C01786=1016.272,-4.523,-107.561,165.907,56.425,160.161
C01787=1016.266,-4.773,-107.549,165.903,56.433,160.162
C01788=1016.261,-5.023,-107.536,165.902,56.442,160.163
C01789=1016.255,-5.301,-107.522,165.899,56.451,160.164
C01790=1016.250,-5.580,-107.508,165.896,56.459,160.165
C01791=1016.243,-5.858,-107.494,165.893,56.468,160.166
C01792=1016.237,-6.136,-107.480,165.889,56.476,160.166
C01793=1016.232,-6.386,-107.466,165.887,56.484,160.167
C01794=1016.226,-6.636,-107.454,165.885,56.492,160.168
C01795=1016.221,-6.886,-107.441,165.882,56.500,160.169
C01796=1016.216,-7.135,-107.429,165.880,56.507,160.170
C01797=1016.210,-7.385,-107.416,165.877,56.515,160.171
C01798=1016.205,-7.634,-107.404,165.874,56.523,160.171
C01799=1016.200,-7.884,-107.391,165.871,56.531,160.172
C01800=1016.194,-8.133,-107.379,165.869,56.538,160.173
C01801=1016.190,-8.384,-107.367,165.866,56.546,160.174
C01802=1016.184,-8.633,-107.354,165.864,56.553,160.175
C01803=1016.179,-8.883,-107.341,165.860,56.561,160.175
C01804=1016.173,-9.133,-107.329,165.858,56.569,160.176
C01805=1016.168,-9.382,-107.317,165.855,56.577,160.177
C01806=1016.164,-9.631,-107.304,165.853,56.584,160.178
C01807=1016.158,-9.881,-107.291,165.850,56.592,160.179
C01808=1016.152,-10.131,-107.279,165.848,56.600,160.180
C01809=1016.147,-10.381,-107.266,165.845,56.607,160.181
C01810=1016.142,-10.630,-107.254,165.842,56.615,160.181
C01811=1016.137,-10.879,-107.242,165.839,56.623,160.182
C01812=1016.131,-11.129,-107.229,165.837,56.630,160.183
C01813=1016.126,-11.379,-107.217,165.834,56.638,160.184
C01814=1016.121,-11.629,-107.204,165.832,56.646,160.185
C01815=1016.116,-11.878,-107.192,165.830,56.653,160.185
C01816=1016.111,-12.128,-107.180,165.827,56.661,160.186
C01817=1016.105,-12.378,-107.166,165.824,56.669,160.187
C01818=1016.100,-12.627,-107.154,165.821,56.677,160.188
C01819=1016.095,-12.876,-107.142,165.819,56.684,160.189
C01820=1016.090,-13.127,-107.130,165.816,56.691,160.189
C01821=1016.085,-13.376,-107.117,165.813,56.699,160.190
C01822=1016.079,-13.625,-107.105,165.811,56.706,160.191
C01823=1016.074,-13.876,-107.092,165.808,56.714,160.192
C01824=1016.069,-14.125,-107.080,165.806,56.722,160.192
C01825=1016.064,-14.374,-107.067,165.803,56.729,160.193
C01826=1016.059,-14.625,-107.055,165.801,56.737,160.194
C01827=1016.053,-14.874,-107.043,165.797,56.744,160.195
C01828=1016.049,-15.123,-107.030,165.795,56.752,160.195
C01829=1016.043,-15.373,-107.018,165.792,56.760,160.196
C01830=1016.038,-15.623,-107.006,165.790,56.767,160.197
C01831=1016.033,-15.873,-106.993,165.787,56.775,160.198
C01832=1016.027,-16.122,-106.981,165.784,56.782,160.198
C01833=1016.022,-16.372,-106.969,165.782,56.790,160.199
C01834=1016.017,-16.621,-106.957,165.779,56.797,160.200
C01835=1016.011,-16.871,-106.945,165.776,56.805,160.201
C01836=1016.006,-17.121,-106.933,165.773,56.813,160.202
C01837=1016.002,-17.371,-106.920,165.771,56.821,160.202
C01838=1015.996,-17.621,-106.909,165.769,56.828,160.203
C01839=1015.991,-17.870,-106.896,165.766,56.836,160.204
C01840=1015.985,-18.120,-106.884,165.764,56.844,160.205
C01841=1015.980,-18.369,-106.873,165.760,56.852,160.206
C01842=1015.975,-18.619,-106.860,165.758,56.859,160.207
C01843=1015.970,-18.869,-106.849,165.755,56.867,160.207
C01844=1015.964,-19.118,-106.837,165.753,56.875,160.208
C01845=1015.959,-19.368,-106.825,165.751,56.882,160.209
C01846=1015.953,-19.618,-106.812,165.747,56.890,160.210
C01847=1015.948,-19.868,-106.801,165.744,56.897,160.210
C01848=1015.943,-20.117,-106.789,165.742,56.905,160.211
C01849=1015.939,-20.367,-106.777,165.739,56.913,160.212
C01850=1015.933,-20.616,-106.765,165.737,56.920,160.213
C01851=1015.928,-20.867,-106.753,165.734,56.928,160.214
C01852=1015.923,-21.116,-106.741,165.732,56.936,160.215
C01853=1015.917,-21.392,-106.727,165.729,56.944,160.215
C01854=1015.911,-21.670,-106.714,165.726,56.952,160.216
C01855=1015.905,-21.946,-106.701,165.722,56.961,160.217
C01856=1015.900,-22.223,-106.688,165.719,56.969,160.218
C01857=1015.894,-22.472,-106.676,165.717,56.977,160.219
C01858=1015.889,-22.722,-106.664,165.714,56.984,160.219
C01859=1015.884,-22.972,-106.652,165.712,56.992,160.220
C01860=1015.879,-23.222,-106.640,165.709,56.999,160.221
C01861=1015.874,-23.471,-106.629,165.707,57.007,160.222
C01862=1015.868,-23.721,-106.617,165.704,57.014,160.222
C01863=1015.863,-23.970,-106.605,165.701,57.022,160.223
C01864=1015.858,-24.220,-106.593,165.699,57.029,160.224
C01865=1015.852,-24.470,-106.581,165.696,57.037,160.225
C01866=1015.847,-24.719,-106.569,165.693,57.044,160.225
C01867=1015.842,-24.969,-106.557,165.690,57.052,160.226
C01868=1015.838,-25.219,-106.545,165.688,57.060,160.227
C01869=1015.832,-25.468,-106.533,165.685,57.067,160.227
C01870=1015.827,-25.718,-106.522,165.682,57.074,160.228
C01871=1015.822,-25.968,-106.510,165.680,57.082,160.229
C01872=1015.817,-26.217,-106.498,165.677,57.089,160.230
C01873=1015.811,-26.468,-106.486,165.675,57.097,160.230
C01874=1015.806,-26.717,-106.474,165.672,57.104,160.231
C01875=1015.801,-26.967,-106.463,165.669,57.111,160.232
C01876=1015.796,-27.216,-106.451,165.667,57.119,160.233
C01877=1015.791,-27.466,-106.439,165.664,57.126,160.233
C01878=1015.786,-27.715,-106.427,165.662,57.134,160.234
C01879=1015.781,-27.965,-106.416,165.659,57.141,160.235
C01880=1015.776,-28.215,-106.404,165.655,57.149,160.235
C01881=1015.771,-28.465,-106.393,165.653,57.156,160.236
C01882=1015.765,-28.714,-106.382,165.651,57.164,160.237
C01883=1015.760,-28.963,-106.370,165.648,57.172,160.238
C01884=1015.755,-29.213,-106.358,165.645,57.179,160.238
C01885=1015.749,-29.464,-106.347,165.643,57.187,160.239
C01886=1015.744,-29.714,-106.335,165.639,57.195,160.240
C01887=1015.738,-29.963,-106.324,165.637,57.202,160.241
C01888=1015.733,-30.213,-106.313,165.634,57.209,160.241
C01889=1015.728,-30.463,-106.301,165.632,57.217,160.242
C01890=1015.723,-30.712,-106.289,165.629,57.225,160.243
C01891=1015.717,-30.961,-106.278,165.627,57.232,160.244
C01892=1015.712,-31.211,-106.267,165.624,57.239,160.245
C01893=1015.707,-31.461,-106.255,165.621,57.248,160.245
C01894=1015.702,-31.711,-106.244,165.618,57.255,160.246
C01895=1015.697,-31.961,-106.232,165.615,57.262,160.247
C01896=1015.692,-32.210,-106.221,165.613,57.270,160.247
C01897=1015.687,-32.460,-106.210,165.611,57.278,160.248
C01898=1015.682,-32.710,-106.199,165.608,57.285,160.249
C01899=1015.677,-32.959,-106.187,165.605,57.292,160.250
C01900=1015.671,-33.209,-106.176,165.602,57.299,160.250
C01901=1015.666,-33.459,-106.165,165.600,57.307,160.251
C01902=1015.661,-33.709,-106.153,165.597,57.315,160.252
C01903=1015.656,-33.958,-106.142,165.594,57.322,160.252
C01904=1015.650,-34.208,-106.131,165.591,57.330,160.253
C01905=1015.645,-34.458,-106.119,165.589,57.337,160.254
C01906=1015.641,-34.707,-106.108,165.586,57.345,160.255
C01907=1015.636,-34.957,-106.097,165.583,57.352,160.255
C01908=1015.631,-35.206,-106.085,165.581,57.359,160.256
C01909=1015.625,-35.456,-106.074,165.578,57.366,160.257
C01910=1015.620,-35.706,-106.063,165.576,57.374,160.257
C01911=1015.615,-35.955,-106.052,165.573,57.381,160.258
C01912=1015.610,-36.205,-106.040,165.570,57.389,160.259
C01913=1015.604,-36.455,-106.029,165.567,57.396,160.259
C01914=1015.599,-36.705,-106.018,165.565,57.403,160.260
C01915=1015.594,-36.954,-106.006,165.562,57.410,160.261
C01916=1015.589,-37.204,-105.995,165.560,57.418,160.262
C01917=1015.584,-37.445,-105.985,165.557,57.425,160.262
C01918=1015.579,-37.685,-105.973,165.554,57.432,160.263
C01919=1015.575,-37.925,-105.963,165.551,57.439,160.263
C01920=1015.570,-38.166,-105.952,165.549,57.447,160.264
C01921=1015.564,-38.406,-105.941,165.547,57.453,160.265
C01922=1015.560,-38.647,-105.930,165.544,57.460,160.266
C01923=1015.555,-38.887,-105.920,165.541,57.467,160.266
C01924=1015.550,-39.128,-105.908,165.538,57.474,160.267
C01925=1015.545,-39.378,-105.898,165.536,57.482,160.267
C01926=1015.540,-39.627,-105.887,165.533,57.489,160.268
C01927=1015.534,-39.877,-105.876,165.531,57.497,160.269
C01928=1015.529,-40.127,-105.864,165.528,57.504,160.269
C01929=1015.524,-40.376,-105.854,165.526,57.512,160.270
C01930=1015.519,-40.626,-105.843,165.523,57.519,160.271
C01931=1015.514,-40.875,-105.832,165.520,57.526,160.272
C01932=1015.509,-41.126,-105.821,165.517,57.535,160.272
C01933=1015.503,-41.375,-105.810,165.514,57.542,160.273
C01934=1015.499,-41.624,-105.799,165.512,57.549,160.274
C01935=1015.493,-41.874,-105.788,165.509,57.556,160.274
C01936=1015.488,-42.124,-105.778,165.507,57.564,160.275
C01937=1015.483,-42.374,-105.767,165.504,57.571,160.276
C01938=1015.478,-42.624,-105.756,165.501,57.579,160.277
C01939=1015.473,-42.873,-105.746,165.498,57.586,160.277
C01940=1015.468,-43.123,-105.734,165.496,57.593,160.278
C01941=1015.462,-43.373,-105.724,165.493,57.601,160.279
C01942=1015.457,-43.623,-105.712,165.490,57.608,160.279
C01943=1015.452,-43.872,-105.702,165.488,57.615,160.280
C01944=1015.448,-44.122,-105.691,165.484,57.623,160.280
C01945=1015.441,-44.416,-105.678,165.481,57.632,160.281
C01946=1015.435,-44.711,-105.665,165.478,57.640,160.282
C01947=1015.430,-45.005,-105.653,165.475,57.649,160.283
C01948=1015.423,-45.299,-105.640,165.472,57.657,160.284
C01949=1015.418,-45.549,-105.630,165.470,57.665,160.284
C01950=1015.413,-45.798,-105.619,165.467,57.672,160.285
C01951=1015.408,-46.048,-105.608,165.464,57.679,160.286
C01952=1015.403,-46.298,-105.597,165.462,57.687,160.286
C01953=1015.397,-46.548,-105.587,165.459,57.694,160.287
C01954=1015.392,-46.797,-105.576,165.456,57.701,160.288
///RCONF 1,0,0,1,0,0,0,0,0,0,0,0,0,0,0,0,0,0,0,0,0,0,0,0
C01955=1015.388,-47.047,-105.565,165.454,57.708,160.288
C01956=1015.382,-47.297,-105.555,165.451,57.715,160.289
C01957=1015.377,-47.546,-105.543,165.448,57.722,160.290
C01958=1015.372,-47.796,-105.533,165.445,57.729,160.290
C01959=1015.367,-48.046,-105.522,165.443,57.737,160.291
C01960=1015.362,-48.295,-105.512,165.440,57.744,160.292
C01961=1015.357,-48.545,-105.501,165.437,57.751,160.292
C01962=1015.352,-48.795,-105.490,165.434,57.758,160.293
C01963=1015.348,-49.045,-105.480,165.432,57.766,160.294
C01964=1015.342,-49.294,-105.469,165.429,57.773,160.294
C01965=1015.337,-49.544,-105.458,165.426,57.780,160.295
C01966=1015.332,-49.793,-105.448,165.423,57.787,160.295
C01967=1015.327,-50.044,-105.437,165.420,57.794,160.296
C01968=1015.322,-50.293,-105.426,165.418,57.802,160.297
C01969=1015.318,-50.543,-105.416,165.415,57.809,160.297
C01970=1015.312,-50.792,-105.405,165.412,57.816,160.298
C01971=1015.307,-51.043,-105.394,165.409,57.823,160.298
C01972=1015.302,-51.292,-105.384,165.407,57.830,160.299
C01973=1015.297,-51.542,-105.374,165.404,57.838,160.300
C01974=1015.291,-51.792,-105.363,165.402,57.845,160.300
C01975=1015.286,-52.041,-105.354,165.399,57.853,160.301
C01976=1015.281,-52.291,-105.343,165.396,57.860,160.302
C01977=1015.275,-52.541,-105.333,165.394,57.868,160.303
C01978=1015.271,-52.791,-105.323,165.391,57.875,160.303
C01979=1015.265,-53.041,-105.313,165.388,57.882,160.304
C01980=1015.260,-53.290,-105.303,165.386,57.889,160.305
C01981=1015.255,-53.566,-105.292,165.383,57.898,160.305
C01982=1015.249,-53.842,-105.280,165.380,57.906,160.306
C01983=1015.243,-54.118,-105.270,165.376,57.914,160.306
C01984=1015.238,-54.394,-105.258,165.374,57.922,160.307
C01985=1015.232,-54.644,-105.248,165.371,57.929,160.308
C01986=1015.227,-54.894,-105.238,165.367,57.936,160.308
C01987=1015.222,-55.144,-105.228,165.365,57.944,160.309
C01988=1015.217,-55.394,-105.218,165.362,57.951,160.310
C01989=1015.212,-55.643,-105.208,165.359,57.958,160.310
C01990=1015.206,-55.894,-105.198,165.357,57.966,160.311
C01991=1015.201,-56.143,-105.188,165.354,57.973,160.312
C01992=1015.196,-56.393,-105.178,165.351,57.980,160.312
C01993=1015.191,-56.642,-105.167,165.349,57.987,160.313
C01994=1015.185,-56.892,-105.157,165.346,57.995,160.314
C01995=1015.181,-57.141,-105.147,165.343,58.002,160.314
C01996=1015.175,-57.391,-105.137,165.341,58.009,160.315
C01997=1015.170,-57.641,-105.127,165.338,58.016,160.315
C01998=1015.165,-57.891,-105.117,165.335,58.023,160.316
C01999=1015.160,-58.140,-105.107,165.333,58.031,160.317
C02000=1015.155,-58.391,-105.096,165.330,58.038,160.317
C02001=1015.151,-58.640,-105.087,165.327,58.045,160.318
C02002=1015.146,-58.890,-105.077,165.324,58.052,160.318
C02003=1015.140,-59.140,-105.067,165.321,58.059,160.319
C02004=1015.135,-59.389,-105.057,165.319,58.067,160.320
C02005=1015.130,-59.639,-105.047,165.316,58.074,160.320
C02006=1015.125,-59.889,-105.037,165.314,58.081,160.321
C02007=1015.120,-60.139,-105.027,165.311,58.088,160.322
C02008=1015.115,-60.388,-105.017,165.308,58.096,160.322
C02009=1015.109,-60.638,-105.007,165.305,58.103,160.323
C02010=1015.105,-60.888,-104.997,165.302,58.110,160.323
C02011=1015.100,-61.137,-104.987,165.299,58.117,160.324
C02012=1015.095,-61.388,-104.978,165.298,58.123,160.325
C02013=1015.090,-61.637,-104.968,165.295,58.130,160.325
C02014=1015.084,-61.887,-104.958,165.292,58.138,160.326
C02015=1015.080,-62.137,-104.948,165.289,58.145,160.326
C02016=1015.075,-62.386,-104.938,165.286,58.152,160.327
C02017=1015.069,-62.636,-104.928,165.284,58.159,160.327
C02018=1015.064,-62.886,-104.918,165.281,58.166,160.328
C02019=1015.059,-63.136,-104.908,165.278,58.173,160.328
C02020=1015.054,-63.385,-104.898,165.275,58.180,160.329
C02021=1015.049,-63.635,-104.889,165.272,58.187,160.330
C02022=1015.044,-63.885,-104.879,165.270,58.194,160.330
C02023=1015.039,-64.135,-104.869,165.268,58.201,160.331
C02024=1015.035,-64.384,-104.860,165.265,58.208,160.331
C02025=1015.029,-64.634,-104.849,165.262,58.215,160.332
C02026=1015.024,-64.884,-104.840,165.259,58.222,160.333
C02027=1015.019,-65.133,-104.830,165.257,58.229,160.333
C02028=1015.015,-65.384,-104.820,165.254,58.236,160.334
C02029=1015.010,-65.633,-104.810,165.251,58.243,160.334
C02030=1015.005,-65.883,-104.800,165.249,58.249,160.335
C02031=1015.000,-66.133,-104.790,165.246,58.256,160.335
C02032=1014.995,-66.382,-104.780,165.243,58.263,160.336
C02033=1014.991,-66.632,-104.771,165.240,58.270,160.336
C02034=1014.986,-66.882,-104.761,165.238,58.278,160.337
C02035=1014.980,-67.132,-104.751,165.235,58.285,160.338
C02036=1014.976,-67.381,-104.741,165.232,58.291,160.338
C02037=1014.971,-67.631,-104.732,165.230,58.298,160.339
C02038=1014.966,-67.882,-104.722,165.227,58.305,160.339
C02039=1014.961,-68.131,-104.712,165.224,58.312,160.340
C02040=1014.956,-68.380,-104.703,165.221,58.319,160.340
C02041=1014.951,-68.630,-104.693,165.219,58.325,160.341
C02042=1014.946,-68.880,-104.683,165.216,58.332,160.341
C02043=1014.941,-69.130,-104.673,165.213,58.339,160.342
C02044=1014.936,-69.379,-104.664,165.210,58.345,160.342
C02045=1014.931,-69.656,-104.653,165.208,58.353,160.343
C02046=1014.926,-69.934,-104.642,165.205,58.360,160.343
C02047=1014.920,-70.210,-104.632,165.201,58.368,160.344
C02048=1014.914,-70.488,-104.621,165.199,58.376,160.345
C02049=1014.909,-70.738,-104.612,165.196,58.382,160.345
C02050=1014.905,-70.987,-104.602,165.193,58.389,160.346
C02051=1014.900,-71.237,-104.592,165.191,58.396,160.346
C02052=1014.895,-71.487,-104.583,165.188,58.402,160.347
C02053=1014.890,-71.737,-104.573,165.185,58.409,160.347
C02054=1014.885,-71.987,-104.564,165.183,58.416,160.348
C02055=1014.881,-72.236,-104.554,165.180,58.422,160.348
C02056=1014.876,-72.486,-104.544,165.177,58.430,160.349
C02057=1014.871,-72.736,-104.535,165.175,58.435,160.349
C02058=1014.866,-72.986,-104.525,165.172,58.443,160.350
C02059=1014.861,-73.235,-104.515,165.169,58.450,160.350
C02060=1014.856,-73.485,-104.506,165.166,58.456,160.350
C02061=1014.852,-73.735,-104.496,165.164,58.463,160.351
C02062=1014.847,-73.985,-104.487,165.161,58.469,160.352
C02063=1014.842,-74.234,-104.477,165.159,58.476,160.352
C02064=1014.837,-74.483,-104.468,165.156,58.482,160.353
C02065=1014.832,-74.734,-104.458,165.153,58.489,160.353
C02066=1014.828,-74.984,-104.449,165.149,58.496,160.353
C02067=1014.823,-75.234,-104.439,165.148,58.502,160.354
C02068=1014.818,-75.484,-104.430,165.145,58.509,160.355
C02069=1014.813,-75.733,-104.421,165.142,58.517,160.355
C02070=1014.808,-75.983,-104.412,165.139,58.523,160.355
C02071=1014.804,-76.233,-104.403,165.137,58.530,160.356
C02072=1014.798,-76.482,-104.394,165.134,58.537,160.357
C02073=1014.794,-76.732,-104.385,165.131,58.543,160.357
C02074=1014.789,-76.982,-104.376,165.128,58.550,160.358
C02075=1014.783,-77.232,-104.366,165.126,58.557,160.358
C02076=1014.778,-77.482,-104.357,165.123,58.563,160.359
C02077=1014.774,-77.732,-104.348,165.120,58.570,160.359
C02078=1014.769,-77.981,-104.338,165.117,58.577,160.359
C02079=1014.764,-78.231,-104.330,165.115,58.583,160.360
C02080=1014.759,-78.481,-104.320,165.113,58.591,160.361
C02081=1014.754,-78.730,-104.311,165.109,58.597,160.361
C02082=1014.749,-78.980,-104.302,165.107,58.604,160.362
C02083=1014.745,-79.230,-104.293,165.104,58.610,160.362
C02084=1014.740,-79.480,-104.284,165.101,58.617,160.363
C02085=1014.735,-79.729,-104.275,165.098,58.624,160.363
C02086=1014.730,-79.979,-104.266,165.096,58.630,160.364
C02087=1014.725,-80.229,-104.257,165.093,58.637,160.364
C02088=1014.721,-80.479,-104.248,165.090,58.644,160.364
C02089=1014.716,-80.729,-104.239,165.089,58.650,160.365
C02090=1014.710,-80.979,-104.231,165.085,58.657,160.365
C02091=1014.706,-81.229,-104.222,165.082,58.664,160.366
C02092=1014.700,-81.478,-104.212,165.080,58.671,160.367
C02093=1014.696,-81.728,-104.203,165.076,58.677,160.367
C02094=1014.691,-81.977,-104.195,165.075,58.684,160.368
C02095=1014.685,-82.227,-104.186,165.072,58.691,160.368
C02096=1014.681,-82.477,-104.177,165.068,58.698,160.368
C02097=1014.675,-82.727,-104.169,165.066,58.705,160.369
C02098=1014.671,-82.977,-104.160,165.063,58.711,160.369
C02099=1014.666,-83.227,-104.151,165.061,58.718,160.370
C02100=1014.661,-83.477,-104.142,165.058,58.725,160.371
C02101=1014.656,-83.726,-104.134,165.056,58.731,160.371
C02102=1014.651,-83.976,-104.125,165.053,58.738,160.372
C02103=1014.646,-84.226,-104.116,165.050,58.745,160.372
C02104=1014.641,-84.476,-104.108,165.047,58.752,160.372
C02105=1014.636,-84.726,-104.098,165.045,58.758,160.373
C02106=1014.632,-84.975,-104.090,165.042,58.765,160.373
C02107=1014.626,-85.225,-104.082,165.038,58.771,160.374
C02108=1014.622,-85.475,-104.073,165.037,58.778,160.374
C02109=1014.616,-85.754,-104.063,165.033,58.786,160.375
C02110=1014.611,-86.033,-104.053,165.030,58.793,160.375
C02111=1014.605,-86.312,-104.044,165.028,58.800,160.376
C02112=1014.600,-86.591,-104.034,165.024,58.807,160.376
C02113=1014.595,-86.841,-104.025,165.022,58.814,160.377
C02114=1014.590,-87.091,-104.017,165.019,58.821,160.377
C02115=1014.585,-87.341,-104.009,165.015,58.827,160.377
C02116=1014.581,-87.590,-104.000,165.014,58.834,160.378
C02117=1014.576,-87.840,-103.992,165.010,58.840,160.378
C02118=1014.571,-88.090,-103.983,165.009,58.847,160.379
C02119=1014.566,-88.340,-103.974,165.005,58.853,160.379
C02120=1014.561,-88.590,-103.966,165.002,58.860,160.380
C02121=1014.556,-88.840,-103.956,165.000,58.866,160.380
C02122=1014.551,-89.089,-103.948,164.997,58.873,160.381
C02123=1014.547,-89.339,-103.939,164.995,58.879,160.381
C02124=1014.542,-89.589,-103.932,164.992,58.886,160.382
C02125=1014.537,-89.839,-103.923,164.990,58.892,160.382
C02126=1014.532,-90.089,-103.914,164.986,58.898,160.382
C02127=1014.527,-90.338,-103.906,164.983,58.905,160.383
C02128=1014.523,-90.588,-103.897,164.981,58.911,160.383
C02129=1014.518,-90.837,-103.888,164.978,58.918,160.384
C02130=1014.513,-91.088,-103.881,164.976,58.924,160.384
C02131=1014.508,-91.338,-103.871,164.973,58.930,160.384
C02132=1014.504,-91.587,-103.863,164.971,58.937,160.385
C02133=1014.499,-91.837,-103.854,164.968,58.943,160.385
C02134=1014.494,-92.087,-103.846,164.965,58.949,160.386
C02135=1014.489,-92.337,-103.838,164.962,58.956,160.386
C02136=1014.485,-92.586,-103.829,164.960,58.962,160.387
C02137=1014.480,-92.836,-103.821,164.957,58.969,160.387
C02138=1014.475,-93.086,-103.812,164.955,58.975,160.388
C02139=1014.470,-93.336,-103.804,164.951,58.981,160.388
C02140=1014.465,-93.585,-103.796,164.949,58.987,160.388
C02141=1014.461,-93.835,-103.787,164.947,58.993,160.389
C02142=1014.456,-94.086,-103.779,164.944,59.000,160.389
C02143=1014.452,-94.335,-103.770,164.941,59.006,160.389
C02144=1014.447,-94.585,-103.762,164.938,59.012,160.390
C02145=1014.442,-94.834,-103.753,164.936,59.018,160.390
C02146=1014.438,-95.084,-103.745,164.933,59.025,160.391
C02147=1014.433,-95.334,-103.737,164.931,59.031,160.391
C02148=1014.427,-95.584,-103.728,164.928,59.037,160.392
C02149=1014.423,-95.834,-103.720,164.925,59.044,160.392
C02150=1014.418,-96.083,-103.712,164.923,59.050,160.392
C02151=1014.414,-96.334,-103.703,164.920,59.056,160.393
C02152=1014.410,-96.583,-103.695,164.917,59.062,160.393
C02153=1014.404,-96.833,-103.687,164.915,59.068,160.393
C02154=1014.400,-97.083,-103.678,164.912,59.074,160.394
C02155=1014.395,-97.333,-103.670,164.909,59.080,160.394
C02156=1014.391,-97.583,-103.661,164.907,59.086,160.395
C02157=1014.386,-97.833,-103.654,164.903,59.092,160.394
C02158=1014.381,-98.082,-103.645,164.901,59.098,160.395
C02159=1014.376,-98.332,-103.638,164.898,59.105,160.396
C02160=1014.372,-98.582,-103.629,164.896,59.111,160.396
C02161=1014.367,-98.832,-103.621,164.893,59.118,160.396
C02162=1014.362,-99.082,-103.613,164.890,59.124,160.397
C02163=1014.357,-99.332,-103.605,164.888,59.130,160.397
C02164=1014.353,-99.581,-103.597,164.885,59.136,160.397
C02165=1014.348,-99.831,-103.589,164.883,59.142,160.398
C02166=1014.343,-100.081,-103.582,164.879,59.149,160.398
C02167=1014.338,-100.331,-103.573,164.877,59.155,160.399
C02168=1014.334,-100.580,-103.566,164.874,59.161,160.399
C02169=1014.328,-100.830,-103.557,164.872,59.167,160.399
C02170=1014.324,-101.081,-103.549,164.869,59.173,160.400
C02171=1014.320,-101.330,-103.541,164.866,59.179,160.400
C02172=1014.315,-101.580,-103.533,164.864,59.185,160.400
C02173=1014.310,-101.861,-103.525,164.861,59.193,160.401
C02174=1014.304,-102.142,-103.516,164.858,59.199,160.401
C02175=1014.299,-102.423,-103.507,164.855,59.206,160.402
C02176=1014.293,-102.704,-103.498,164.852,59.213,160.402
C02177=1014.288,-102.953,-103.490,164.850,59.219,160.402
C02178=1014.284,-103.204,-103.482,164.846,59.225,160.403
C02179=1014.279,-103.453,-103.475,164.844,59.231,160.403
C02180=1014.275,-103.703,-103.466,164.842,59.237,160.404
C02181=1014.270,-103.953,-103.458,164.838,59.244,160.404
C02182=1014.265,-104.203,-103.450,164.836,59.250,160.404
C02183=1014.261,-104.453,-103.443,164.834,59.256,160.405
C02184=1014.256,-104.703,-103.435,164.831,59.262,160.405
C02185=1014.251,-104.952,-103.427,164.828,59.267,160.405
C02186=1014.246,-105.203,-103.419,164.826,59.273,160.405
C02187=1014.242,-105.452,-103.412,164.822,59.280,160.406
C02188=1014.237,-105.702,-103.404,164.820,59.286,160.406
C02189=1014.232,-105.952,-103.396,164.818,59.292,160.407
C02190=1014.228,-106.201,-103.389,164.816,59.298,160.407
C02191=1014.223,-106.452,-103.381,164.812,59.304,160.407
C02192=1014.218,-106.701,-103.373,164.809,59.310,160.407
C02193=1014.213,-106.951,-103.365,164.807,59.316,160.408
C02194=1014.209,-107.201,-103.358,164.805,59.322,160.408
C02195=1014.204,-107.451,-103.350,164.801,59.327,160.408
C02196=1014.200,-107.701,-103.343,164.799,59.333,160.409
C02197=1014.195,-107.950,-103.335,164.797,59.339,160.409
C02198=1014.190,-108.201,-103.327,164.794,59.345,160.410
C02199=1014.186,-108.450,-103.319,164.792,59.351,160.410
C02200=1014.181,-108.700,-103.311,164.788,59.357,160.410
C02201=1014.176,-108.950,-103.304,164.786,59.363,160.410
C02202=1014.172,-109.199,-103.297,164.784,59.369,160.411
C02203=1014.167,-109.450,-103.289,164.781,59.375,160.411
C02204=1014.163,-109.699,-103.281,164.778,59.381,160.411
C02205=1014.158,-109.950,-103.274,164.775,59.387,160.412
C02206=1014.153,-110.199,-103.267,164.773,59.393,160.412
C02207=1014.148,-110.448,-103.259,164.771,59.399,160.413
C02208=1014.143,-110.699,-103.252,164.767,59.405,160.413
C02209=1014.139,-110.948,-103.244,164.765,59.411,160.413
C02210=1014.135,-111.198,-103.237,164.763,59.417,160.413
C02211=1014.130,-111.448,-103.229,164.760,59.422,160.414
C02212=1014.125,-111.698,-103.222,164.757,59.428,160.414
C02213=1014.121,-111.948,-103.214,164.755,59.434,160.415
C02214=1014.115,-112.198,-103.207,164.751,59.440,160.414
C02215=1014.111,-112.447,-103.200,164.749,59.446,160.415
C02216=1014.107,-112.697,-103.192,164.747,59.452,160.415
C02217=1014.102,-112.947,-103.185,164.744,59.457,160.415
C02218=1014.097,-113.197,-103.177,164.742,59.463,160.416
C02219=1014.093,-113.447,-103.170,164.739,59.468,160.416
C02220=1014.089,-113.697,-103.163,164.737,59.474,160.416
C02221=1014.084,-113.947,-103.155,164.734,59.480,160.417
C02222=1014.080,-114.197,-103.148,164.732,59.486,160.417
C02223=1014.075,-114.446,-103.141,164.728,59.492,160.417
C02224=1014.070,-114.696,-103.133,164.726,59.497,160.417
C02225=1014.065,-114.946,-103.126,164.723,59.503,160.418
C02226=1014.061,-115.196,-103.119,164.720,59.509,160.418
C02227=1014.056,-115.445,-103.111,164.718,59.515,160.418
C02228=1014.051,-115.696,-103.105,164.715,59.520,160.419
C02229=1014.047,-115.946,-103.097,164.713,59.526,160.419
C02230=1014.042,-116.195,-103.090,164.710,59.531,160.419
C02231=1014.038,-116.445,-103.082,164.708,59.537,160.420
C02232=1014.032,-116.695,-103.075,164.705,59.543,160.420
C02233=1014.028,-116.945,-103.069,164.703,59.549,160.420
C02234=1014.024,-117.195,-103.061,164.700,59.554,160.420
C02235=1014.020,-117.444,-103.054,164.698,59.560,160.421
C02236=1014.014,-117.694,-103.047,164.695,59.565,160.421
C02237=1014.009,-117.976,-103.039,164.692,59.572,160.421
C02238=1014.004,-118.257,-103.031,164.689,59.578,160.421
C02239=1013.999,-118.538,-103.023,164.686,59.584,160.422
C02240=1013.994,-118.819,-103.015,164.683,59.591,160.422
C02241=1013.989,-119.069,-103.008,164.681,59.597,160.422
C02242=1013.985,-119.320,-103.001,164.678,59.602,160.423
C02243=1013.980,-119.569,-102.994,164.676,59.608,160.423
C02244=1013.975,-119.819,-102.986,164.673,59.613,160.423
C02245=1013.971,-120.069,-102.980,164.670,59.619,160.423
C02246=1013.966,-120.318,-102.973,164.668,59.625,160.424
C02247=1013.962,-120.568,-102.966,164.665,59.630,160.424
C02248=1013.957,-120.819,-102.959,164.663,59.636,160.424
C02249=1013.953,-121.068,-102.951,164.660,59.641,160.424
C02250=1013.948,-121.318,-102.945,164.657,59.647,160.425
C02251=1013.944,-121.568,-102.938,164.655,59.653,160.425
C02252=1013.939,-121.818,-102.930,164.652,59.658,160.425
C02253=1013.935,-122.068,-102.924,164.649,59.663,160.425
C02254=1013.930,-122.317,-102.917,164.648,59.669,160.426
C02255=1013.926,-122.567,-102.910,164.645,59.674,160.426
C02256=1013.921,-122.817,-102.903,164.643,59.679,160.426
C02257=1013.916,-123.067,-102.895,164.640,59.685,160.426
C02258=1013.912,-123.317,-102.889,164.638,59.691,160.427
C02259=1013.907,-123.567,-102.882,164.635,59.696,160.427
C02260=1013.903,-123.817,-102.875,164.632,59.701,160.427
C02261=1013.898,-124.066,-102.868,164.629,59.707,160.427
C02262=1013.894,-124.317,-102.862,164.627,59.711,160.428
C02263=1013.889,-124.566,-102.854,164.625,59.717,160.428
C02264=1013.885,-124.816,-102.848,164.622,59.723,160.428
C02265=1013.880,-125.066,-102.841,164.619,59.728,160.428
C02266=1013.876,-125.316,-102.834,164.617,59.733,160.428
C02267=1013.871,-125.565,-102.827,164.614,59.739,160.429
C02268=1013.867,-125.816,-102.821,164.612,59.745,160.429
C02269=1013.862,-126.066,-102.815,164.609,59.750,160.429
C02270=1013.858,-126.315,-102.807,164.607,59.755,160.429
C02271=1013.853,-126.565,-102.801,164.604,59.760,160.430
C02272=1013.849,-126.815,-102.794,164.602,59.766,160.430
C02273=1013.844,-127.065,-102.788,164.599,59.771,160.430
C02274=1013.840,-127.315,-102.781,164.596,59.777,160.430
C02275=1013.835,-127.564,-102.774,164.595,59.782,160.431
C02276=1013.831,-127.814,-102.767,164.592,59.787,160.431
C02277=1013.826,-128.064,-102.761,164.589,59.792,160.431
C02278=1013.822,-128.314,-102.754,164.586,59.797,160.431
C02279=1013.818,-128.563,-102.747,164.584,59.802,160.431
C02280=1013.813,-128.813,-102.739,164.582,59.806,160.431
C02281=1013.810,-129.062,-102.730,164.580,59.810,160.431
C02282=1013.807,-129.312,-102.721,164.578,59.813,160.431
C02283=1013.804,-129.562,-102.712,164.575,59.817,160.431
C02284=1013.802,-129.812,-102.701,164.572,59.819,160.431
C02285=1013.799,-130.061,-102.690,164.570,59.821,160.430
C02286=1013.798,-130.311,-102.679,164.568,59.821,160.430
C02287=1013.797,-130.560,-102.666,164.566,59.822,160.429
C02288=1013.796,-130.810,-102.653,164.563,59.822,160.429
C02289=1013.795,-131.060,-102.640,164.561,59.822,160.428
C02290=1013.795,-131.310,-102.626,164.560,59.822,160.427
C02291=1013.794,-131.559,-102.612,164.557,59.821,160.426
C02292=1013.795,-131.809,-102.597,164.555,59.819,160.425
C02293=1013.796,-132.059,-102.581,164.552,59.817,160.424
C02294=1013.797,-132.308,-102.565,164.551,59.814,160.423
C02295=1013.798,-132.558,-102.548,164.549,59.811,160.422
C02296=1013.800,-132.807,-102.530,164.547,59.808,160.421
C02297=1013.802,-133.057,-102.512,164.545,59.803,160.419
C02298=1013.804,-133.307,-102.493,164.543,59.799,160.418
C02299=1013.807,-133.556,-102.473,164.541,59.794,160.416
C02300=1013.810,-133.806,-102.453,164.539,59.788,160.415
C02301=1013.579,-133.832,-102.870,164.519,60.110,160.468
C02302=1013.576,-133.583,-102.890,164.521,60.115,160.470
C02303=1013.574,-133.333,-102.909,164.523,60.119,160.471
C02304=1013.571,-133.083,-102.928,164.526,60.124,160.473
C02305=1013.570,-132.833,-102.947,164.527,60.128,160.474
C02306=1013.568,-132.584,-102.965,164.530,60.131,160.475
C02307=1013.566,-132.334,-102.982,164.530,60.134,160.476
C02308=1013.565,-132.084,-102.997,164.533,60.137,160.478
C02309=1013.564,-131.835,-103.014,164.535,60.139,160.478
C02310=1013.564,-131.585,-103.029,164.538,60.140,160.480
C02311=1013.564,-131.336,-103.043,164.539,60.142,160.480
C02312=1013.565,-131.086,-103.057,164.541,60.142,160.481
C02313=1013.565,-130.836,-103.071,164.544,60.142,160.482
C02314=1013.566,-130.587,-103.083,164.545,60.142,160.482
C02315=1013.568,-130.338,-103.096,164.548,60.141,160.483
C02316=1013.569,-130.088,-103.107,164.550,60.140,160.483
C02317=1013.571,-129.838,-103.119,164.552,60.138,160.484
C02318=1013.574,-129.588,-103.129,164.554,60.137,160.484
C02319=1013.576,-129.338,-103.138,164.558,60.134,160.485
C02320=1013.579,-129.088,-103.148,164.560,60.131,160.485
C02321=1013.583,-128.839,-103.156,164.562,60.127,160.485
C02322=1013.586,-128.590,-103.164,164.563,60.123,160.484
C02323=1013.590,-128.340,-103.171,164.567,60.119,160.485
C02324=1013.595,-128.090,-103.178,164.568,60.114,160.484
C02325=1013.600,-127.841,-103.185,164.571,60.109,160.484
C02326=1013.604,-127.591,-103.191,164.574,60.104,160.484
C02327=1013.608,-127.342,-103.198,164.576,60.099,160.484
C02328=1013.613,-127.092,-103.204,164.579,60.094,160.484
C02329=1013.617,-126.842,-103.211,164.581,60.089,160.484
C02330=1013.622,-126.592,-103.218,164.584,60.084,160.483
C02331=1013.626,-126.342,-103.224,164.587,60.078,160.483
C02332=1013.631,-126.092,-103.230,164.588,60.073,160.483
C02333=1013.635,-125.842,-103.238,164.591,60.068,160.483
C02334=1013.640,-125.593,-103.244,164.594,60.063,160.483
C02335=1013.644,-125.342,-103.251,164.597,60.058,160.483
C02336=1013.648,-125.093,-103.258,164.598,60.053,160.482
C02337=1013.653,-124.843,-103.264,164.601,60.047,160.482
C02338=1013.658,-124.593,-103.272,164.604,60.042,160.482
C02339=1013.662,-124.343,-103.278,164.606,60.037,160.482
C02340=1013.667,-124.093,-103.285,164.608,60.032,160.481
C02341=1013.671,-123.843,-103.292,164.611,60.027,160.481
C02342=1013.677,-123.593,-103.299,164.613,60.022,160.481
C02343=1013.681,-123.343,-103.306,164.616,60.016,160.481
C02344=1013.685,-123.093,-103.313,164.619,60.011,160.481
C02345=1013.690,-122.843,-103.319,164.621,60.006,160.481
C02346=1013.694,-122.594,-103.327,164.623,60.001,160.480
C02347=1013.698,-122.343,-103.333,164.626,59.996,160.480
C02348=1013.703,-122.094,-103.340,164.629,59.990,160.480
C02349=1013.707,-121.844,-103.347,164.632,59.985,160.480
C02350=1013.712,-121.594,-103.354,164.633,59.980,160.479
C02351=1013.716,-121.344,-103.360,164.636,59.975,160.479
C02352=1013.721,-121.095,-103.368,164.638,59.969,160.479
C02353=1013.725,-120.845,-103.375,164.641,59.963,160.479
C02354=1013.731,-120.594,-103.381,164.644,59.958,160.479
C02355=1013.735,-120.345,-103.389,164.646,59.953,160.478
C02356=1013.739,-120.095,-103.396,164.648,59.948,160.478
C02357=1013.744,-119.845,-103.402,164.651,59.943,160.478
C02358=1013.748,-119.596,-103.410,164.654,59.937,160.478
C02359=1013.752,-119.345,-103.416,164.656,59.931,160.477
C02360=1013.757,-119.096,-103.424,164.659,59.926,160.477
C02361=1013.762,-118.846,-103.431,164.662,59.921,160.477
C02362=1013.766,-118.565,-103.438,164.664,59.915,160.477
C02363=1013.772,-118.283,-103.447,164.667,59.908,160.476
C02364=1013.778,-118.002,-103.454,164.670,59.903,160.476
C02365=1013.783,-117.721,-103.463,164.673,59.896,160.476
C02366=1013.787,-117.471,-103.470,164.675,59.891,160.476
C02367=1013.792,-117.222,-103.477,164.677,59.885,160.475
C02368=1013.796,-116.972,-103.483,164.680,59.880,160.475
C02369=1013.800,-116.722,-103.491,164.683,59.875,160.475
C02370=1013.805,-116.472,-103.499,164.685,59.869,160.475
C02371=1013.810,-116.222,-103.506,164.688,59.863,160.474
C02372=1013.815,-115.972,-103.512,164.690,59.858,160.474
C02373=1013.819,-115.723,-103.519,164.693,59.853,160.474
C02374=1013.823,-115.473,-103.527,164.695,59.847,160.474
C02375=1013.828,-115.223,-103.535,164.698,59.841,160.473
C02376=1013.833,-114.973,-103.541,164.700,59.835,160.473
C02377=1013.837,-114.723,-103.548,164.703,59.830,160.473
C02378=1013.842,-114.474,-103.556,164.706,59.825,160.473
C02379=1013.847,-114.223,-103.563,164.708,59.819,160.472
C02380=1013.851,-113.974,-103.571,164.711,59.813,160.472
C02381=1013.855,-113.724,-103.578,164.714,59.808,160.472
C02382=1013.860,-113.475,-103.585,164.716,59.802,160.471
C02383=1013.865,-113.224,-103.592,164.719,59.797,160.471
C02384=1013.869,-112.974,-103.599,164.722,59.791,160.471
C02385=1013.874,-112.724,-103.607,164.724,59.785,160.471
C02386=1013.878,-112.475,-103.614,164.727,59.780,160.471
C02387=1013.883,-112.224,-103.622,164.729,59.774,160.470
C02388=1013.887,-111.975,-103.629,164.732,59.769,160.470
C02389=1013.892,-111.725,-103.637,164.734,59.763,160.469
C02390=1013.896,-111.475,-103.644,164.737,59.757,160.469
C02391=1013.902,-111.225,-103.651,164.739,59.751,160.469
C02392=1013.906,-110.976,-103.659,164.742,59.746,160.469
C02393=1013.911,-110.726,-103.666,164.744,59.740,160.468
C02394=1013.916,-110.476,-103.674,164.747,59.735,160.468
C02395=1013.920,-110.226,-103.681,164.749,59.729,160.468
C02396=1013.924,-109.977,-103.689,164.751,59.723,160.468
C02397=1013.929,-109.726,-103.696,164.754,59.717,160.467
C02398=1013.934,-109.477,-103.704,164.756,59.712,160.467
C02399=1013.939,-109.227,-103.711,164.760,59.705,160.467
C02400=1013.944,-108.977,-103.718,164.763,59.700,160.467
C02401=1013.948,-108.727,-103.726,164.765,59.694,160.466
C02402=1013.952,-108.478,-103.733,164.767,59.688,160.466
C02403=1013.957,-108.227,-103.741,164.770,59.683,160.465
C02404=1013.962,-107.978,-103.748,164.772,59.677,160.465
C02405=1013.967,-107.727,-103.756,164.775,59.671,160.465
C02406=1013.971,-107.478,-103.764,164.777,59.665,160.464
C02407=1013.975,-107.228,-103.771,164.780,59.659,160.464
C02408=1013.980,-106.978,-103.779,164.783,59.654,160.464
C02409=1013.985,-106.728,-103.786,164.785,59.648,160.464
C02410=1013.990,-106.478,-103.795,164.788,59.642,160.463
C02411=1013.994,-106.229,-103.802,164.790,59.636,160.463
C02412=1013.999,-105.979,-103.809,164.792,59.630,160.462
C02413=1014.004,-105.729,-103.817,164.795,59.625,160.462
C02414=1014.008,-105.479,-103.825,164.798,59.619,160.462
C02415=1014.013,-105.229,-103.832,164.801,59.612,160.462
C02416=1014.018,-104.980,-103.841,164.803,59.607,160.461
C02417=1014.022,-104.729,-103.849,164.806,59.601,160.461
C02418=1014.026,-104.480,-103.856,164.808,59.595,160.461
C02419=1014.031,-104.230,-103.864,164.812,59.589,160.461
C02420=1014.036,-103.980,-103.872,164.814,59.583,160.460
C02421=1014.040,-103.731,-103.880,164.816,59.577,160.460
C02422=1014.045,-103.480,-103.887,164.818,59.571,160.459
C02423=1014.049,-103.231,-103.895,164.821,59.566,160.459
C02424=1014.055,-102.981,-103.903,164.824,59.560,160.459
C02425=1014.059,-102.731,-103.911,164.827,59.554,160.458
C02426=1014.065,-102.450,-103.920,164.830,59.547,160.458
C02427=1014.070,-102.169,-103.928,164.832,59.540,160.458
C02428=1014.075,-101.889,-103.937,164.836,59.533,160.457
C02429=1014.081,-101.607,-103.946,164.839,59.527,160.457
C02430=1014.084,-101.357,-103.954,164.841,59.521,160.457
C02431=1014.089,-101.107,-103.962,164.843,59.515,160.456
C02432=1014.094,-100.858,-103.970,164.846,59.509,160.456
C02433=1014.099,-100.608,-103.978,164.849,59.502,160.455
C02434=1014.103,-100.358,-103.985,164.851,59.496,160.455
C02435=1014.109,-100.108,-103.994,164.854,59.491,160.455
C02436=1014.113,-99.859,-104.001,164.857,59.485,160.455
C02437=1014.118,-99.609,-104.010,164.859,59.478,160.454
C02438=1014.123,-99.359,-104.017,164.861,59.472,160.454
C02439=1014.128,-99.109,-104.025,164.865,59.466,160.453
C02440=1014.132,-98.859,-104.034,164.867,59.460,160.453
C02441=1014.136,-98.609,-104.041,164.869,59.454,160.452
C02442=1014.141,-98.359,-104.049,164.872,59.447,160.452
C02443=1014.146,-98.110,-104.057,164.875,59.441,160.452
C02444=1014.151,-97.860,-104.065,164.878,59.435,160.451
C02445=1014.156,-97.610,-104.074,164.880,59.429,160.451
C02446=1014.160,-97.360,-104.082,164.883,59.424,160.451
C02447=1014.165,-97.110,-104.090,164.885,59.418,160.450
C02448=1014.169,-96.861,-104.099,164.888,59.411,160.450
C02449=1014.174,-96.611,-104.107,164.891,59.405,160.450
C02450=1014.179,-96.361,-104.116,164.893,59.399,160.449
C02451=1014.183,-96.111,-104.123,164.896,59.393,160.449
C02452=1014.188,-95.861,-104.132,164.898,59.387,160.448
C02453=1014.193,-95.611,-104.141,164.901,59.381,160.448
C02454=1014.197,-95.362,-104.148,164.903,59.375,160.448
C02455=1014.202,-95.112,-104.156,164.907,59.369,160.448
C02456=1014.207,-94.862,-104.166,164.909,59.363,160.447
C02457=1014.211,-94.612,-104.173,164.911,59.357,160.447
C02458=1014.216,-94.362,-104.182,164.914,59.350,160.446
C02459=1014.221,-94.113,-104.191,164.917,59.344,160.446
C02460=1014.225,-93.863,-104.198,164.920,59.338,160.446
C02461=1014.230,-93.613,-104.207,164.922,59.332,160.445
C02462=1014.235,-93.363,-104.215,164.924,59.326,160.445
C02463=1014.239,-93.113,-104.223,164.928,59.320,160.445
C02464=1014.244,-92.864,-104.232,164.930,59.314,160.444
C02465=1014.249,-92.614,-104.240,164.933,59.307,160.444
C02466=1014.253,-92.365,-104.249,164.935,59.301,160.443
C02467=1014.258,-92.114,-104.257,164.937,59.295,160.443
C02468=1014.263,-91.864,-104.266,164.941,59.289,160.443
C02469=1014.268,-91.614,-104.275,164.943,59.283,160.442
C02470=1014.273,-91.365,-104.283,164.946,59.276,160.442
C02471=1014.277,-91.115,-104.291,164.948,59.269,160.441
C02472=1014.282,-90.865,-104.299,164.951,59.263,160.441
C02473=1014.286,-90.616,-104.308,164.953,59.257,160.440
C02474=1014.291,-90.366,-104.317,164.957,59.251,160.440
C02475=1014.296,-90.116,-104.324,164.959,59.245,160.440
C02476=1014.301,-89.866,-104.334,164.962,59.238,160.439
C02477=1014.306,-89.617,-104.342,164.964,59.232,160.439
C02478=1014.310,-89.367,-104.351,164.967,59.225,160.438
C02479=1014.315,-89.117,-104.359,164.969,59.219,160.438
C02480=1014.320,-88.867,-104.367,164.973,59.212,160.438
C02481=1014.325,-88.617,-104.376,164.975,59.206,160.437
C02482=1014.329,-88.368,-104.384,164.977,59.199,160.437
C02483=1014.334,-88.118,-104.393,164.980,59.193,160.436
C02484=1014.339,-87.868,-104.402,164.983,59.187,160.436
C02485=1014.344,-87.618,-104.410,164.985,59.181,160.435
C02486=1014.349,-87.367,-104.419,164.988,59.174,160.435
C02487=1014.353,-87.118,-104.427,164.990,59.168,160.434
C02488=1014.358,-86.868,-104.436,164.993,59.161,160.434
C02489=1014.363,-86.619,-104.444,164.996,59.154,160.434
C02490=1014.368,-86.340,-104.454,164.999,59.148,160.433
C02491=1014.374,-86.060,-104.464,165.002,59.140,160.433
C02492=1014.380,-85.782,-104.473,165.005,59.133,160.432
C02493=1014.385,-85.503,-104.483,165.008,59.126,160.432
C02494=1014.390,-85.253,-104.491,165.010,59.119,160.431
C02495=1014.395,-85.003,-104.500,165.013,59.112,160.431
C02496=1014.400,-84.754,-104.509,165.016,59.105,160.430
C02497=1014.404,-84.504,-104.518,165.018,59.099,160.430
C02498=1014.409,-84.255,-104.526,165.022,59.093,160.429
C02499=1014.414,-84.005,-104.535,165.023,59.086,160.429
C02500=1014.419,-83.755,-104.543,165.026,59.080,160.428
C02501=1014.424,-83.505,-104.552,165.029,59.072,160.428
C02502=1014.429,-83.255,-104.561,165.031,59.066,160.427
C02503=1014.434,-83.005,-104.569,165.034,59.059,160.427
C02504=1014.438,-82.755,-104.578,165.037,59.053,160.427
C02505=1014.444,-82.506,-104.587,165.040,59.046,160.426
C02506=1014.449,-82.256,-104.595,165.042,59.040,160.425
C02507=1014.453,-82.006,-104.605,165.045,59.033,160.425
C02508=1014.459,-81.756,-104.613,165.048,59.026,160.425
C02509=1014.463,-81.507,-104.622,165.050,59.019,160.424
C02510=1014.468,-81.257,-104.630,165.053,59.012,160.423
C02511=1014.472,-81.007,-104.639,165.056,59.006,160.423
C02512=1014.478,-80.757,-104.648,165.059,58.999,160.422
C02513=1014.483,-80.508,-104.656,165.061,58.993,160.422
C02514=1014.488,-80.258,-104.665,165.063,58.985,160.421
C02515=1014.492,-80.008,-104.674,165.067,58.979,160.421
C02516=1014.497,-79.758,-104.683,165.068,58.972,160.420
C02517=1014.502,-79.508,-104.692,165.072,58.966,160.420
C02518=1014.507,-79.259,-104.702,165.074,58.959,160.420
C02519=1014.511,-79.008,-104.711,165.077,58.953,160.419
C02520=1014.516,-78.759,-104.719,165.080,58.946,160.419
C02521=1014.521,-78.509,-104.728,165.083,58.939,160.418
C02522=1014.526,-78.259,-104.738,165.085,58.933,160.418
C02523=1014.531,-78.010,-104.747,165.088,58.926,160.417
C02524=1014.536,-77.760,-104.756,165.091,58.920,160.417
C02525=1014.540,-77.510,-104.765,165.093,58.913,160.416
C02526=1014.546,-77.260,-104.774,165.095,58.906,160.416
C02527=1014.551,-77.010,-104.783,165.099,58.899,160.415
C02528=1014.555,-76.760,-104.793,165.100,58.893,160.415
C02529=1014.560,-76.510,-104.802,165.104,58.886,160.414
C02530=1014.565,-76.261,-104.811,165.106,58.879,160.414
C02531=1014.570,-76.011,-104.820,165.110,58.873,160.413
C02532=1014.575,-75.761,-104.830,165.111,58.866,160.413
C02533=1014.580,-75.511,-104.838,165.114,58.859,160.412
C02534=1014.585,-75.261,-104.847,165.117,58.852,160.412
C02535=1014.589,-75.012,-104.857,165.120,58.845,160.411
C02536=1014.595,-74.762,-104.866,165.122,58.838,160.410
C02537=1014.599,-74.512,-104.875,165.125,58.832,160.410
C02538=1014.604,-74.263,-104.884,165.128,58.825,160.410
C02539=1014.609,-74.013,-104.894,165.130,58.819,160.409
C02540=1014.614,-73.763,-104.904,165.133,58.812,160.409
C02541=1014.619,-73.513,-104.913,165.136,58.805,160.408
C02542=1014.623,-73.263,-104.923,165.138,58.799,160.408
C02543=1014.628,-73.014,-104.932,165.141,58.792,160.407
C02544=1014.633,-72.764,-104.941,165.143,58.786,160.407
C02545=1014.638,-72.514,-104.951,165.146,58.779,160.406
C02546=1014.642,-72.264,-104.960,165.149,58.772,160.406
C02547=1014.647,-72.015,-104.970,165.152,58.766,160.405
C02548=1014.652,-71.764,-104.980,165.154,58.759,160.405
C02549=1014.657,-71.515,-104.989,165.157,58.753,160.404
C02550=1014.662,-71.265,-104.999,165.160,58.745,160.404
C02551=1014.666,-71.015,-105.008,165.162,58.739,160.403
C02552=1014.671,-70.766,-105.018,165.165,58.732,160.403
C02553=1014.676,-70.517,-105.028,165.167,58.725,160.402
C02554=1014.681,-70.239,-105.039,165.170,58.718,160.402
C02555=1014.687,-69.962,-105.050,165.173,58.711,160.401
C02556=1014.692,-69.685,-105.060,165.177,58.703,160.401
C02557=1014.697,-69.409,-105.071,165.179,58.695,160.400
C02558=1014.701,-69.159,-105.080,165.182,58.689,160.399
C02559=1014.707,-68.908,-105.090,165.185,58.682,160.399
C02560=1014.712,-68.659,-105.100,165.186,58.675,160.398
C02561=1014.716,-68.409,-105.109,165.190,58.669,160.398
C02562=1014.721,-68.160,-105.119,165.193,58.662,160.397
C02563=1014.726,-67.909,-105.129,165.195,58.655,160.397
C02564=1014.731,-67.659,-105.138,165.198,58.649,160.396
C02565=1014.736,-67.410,-105.148,165.200,58.642,160.396
C02566=1014.741,-67.161,-105.158,165.203,58.634,160.395
C02567=1014.745,-66.911,-105.167,165.206,58.627,160.395
C02568=1014.751,-66.661,-105.177,165.209,58.620,160.394
C02569=1014.755,-66.411,-105.187,165.211,58.614,160.393
C02570=1014.760,-66.162,-105.196,165.214,58.607,160.393
C02571=1014.766,-65.912,-105.207,165.216,58.600,160.392
C02572=1014.770,-65.662,-105.216,165.219,58.593,160.392
C02573=1014.775,-65.412,-105.226,165.222,58.586,160.391
C02574=1014.780,-65.163,-105.235,165.225,58.579,160.391
C02575=1014.785,-64.913,-105.245,165.227,58.573,160.390
C02576=1014.790,-64.663,-105.255,165.230,58.566,160.390
C02577=1014.795,-64.413,-105.264,165.232,58.558,160.389
C02578=1014.800,-64.163,-105.275,165.235,58.551,160.388
C02579=1014.805,-63.914,-105.284,165.238,58.544,160.388
C02580=1014.810,-63.664,-105.294,165.240,58.537,160.387
C02581=1014.815,-63.414,-105.304,165.243,58.530,160.387
C02582=1014.820,-63.164,-105.313,165.246,58.523,160.386
C02583=1014.825,-62.915,-105.323,165.248,58.516,160.385
C02584=1014.830,-62.665,-105.333,165.250,58.509,160.385
C02585=1014.835,-62.415,-105.343,165.254,58.503,160.384
C02586=1014.840,-62.166,-105.353,165.257,58.496,160.384
C02587=1014.844,-61.915,-105.363,165.259,58.488,160.383
C02588=1014.849,-61.665,-105.373,165.262,58.481,160.383
C02589=1014.854,-61.416,-105.383,165.265,58.474,160.382
C02590=1014.859,-61.166,-105.393,165.268,58.467,160.382
C02591=1014.864,-60.916,-105.402,165.270,58.459,160.381
C02592=1014.869,-60.667,-105.412,165.272,58.452,160.380
C02593=1014.874,-60.417,-105.422,165.275,58.445,160.380
C02594=1014.879,-60.168,-105.432,165.278,58.438,160.379
C02595=1014.884,-59.917,-105.442,165.281,58.431,160.378
C02596=1014.889,-59.668,-105.452,165.284,58.424,160.378
C02597=1014.894,-59.418,-105.461,165.286,58.417,160.377
C02598=1014.899,-59.168,-105.471,165.289,58.409,160.377
C02599=1014.904,-58.918,-105.481,165.292,58.402,160.376
C02600=1014.910,-58.668,-105.491,165.295,58.395,160.376
C02601=1014.914,-58.419,-105.501,165.297,58.388,160.375
C02602=1014.919,-58.170,-105.511,165.299,58.380,160.374
C02603=1014.925,-57.919,-105.521,165.302,58.373,160.374
C02604=1014.929,-57.670,-105.531,165.305,58.366,160.373
C02605=1014.935,-57.420,-105.541,165.308,58.359,160.372
C02606=1014.940,-57.170,-105.551,165.311,58.352,160.372
C02607=1014.945,-56.920,-105.561,165.313,58.345,160.371
C02608=1014.950,-56.671,-105.571,165.315,58.337,160.370
C02609=1014.955,-56.421,-105.581,165.318,58.330,160.370
C02610=1014.960,-56.171,-105.591,165.321,58.323,160.369
C02611=1014.966,-55.921,-105.601,165.324,58.316,160.369
C02612=1014.970,-55.672,-105.611,165.326,58.308,160.368
C02613=1014.975,-55.422,-105.622,165.329,58.301,160.367
C02614=1014.980,-55.172,-105.631,165.332,58.294,160.367
C02615=1014.986,-54.922,-105.641,165.334,58.287,160.366
C02616=1014.990,-54.673,-105.651,165.336,58.279,160.365
C02617=1014.996,-54.422,-105.661,165.339,58.272,160.365
C02618=1015.001,-54.148,-105.672,165.343,58.263,160.364
C02619=1015.007,-53.872,-105.684,165.346,58.255,160.363
C02620=1015.013,-53.596,-105.694,165.348,58.247,160.362
C02621=1015.019,-53.320,-105.706,165.351,58.239,160.362
C02622=1015.023,-53.070,-105.716,165.354,58.232,160.361
C02623=1015.029,-52.820,-105.726,165.356,58.224,160.360
C02624=1015.034,-52.570,-105.736,165.360,58.217,160.360
C02625=1015.039,-52.321,-105.746,165.362,58.209,160.359
C02626=1015.044,-52.070,-105.756,165.365,58.202,160.358
C02627=1015.049,-51.821,-105.766,165.368,58.195,160.358
C02628=1015.055,-51.572,-105.777,165.370,58.187,160.357
C02629=1015.060,-51.322,-105.787,165.373,58.180,160.356
C02630=1015.065,-51.072,-105.797,165.375,58.172,160.355
C02631=1015.070,-50.822,-105.808,165.378,58.165,160.355
C02632=1015.074,-50.573,-105.819,165.381,58.158,160.354
C02633=1015.080,-50.322,-105.829,165.383,58.151,160.354
C02634=1015.085,-50.072,-105.840,165.386,58.144,160.353
C02635=1015.090,-49.823,-105.850,165.389,58.137,160.353
C02636=1015.094,-49.573,-105.861,165.391,58.129,160.352
C02637=1015.100,-49.324,-105.871,165.394,58.122,160.351
C02638=1015.104,-49.074,-105.882,165.397,58.115,160.351
C02639=1015.110,-48.823,-105.892,165.400,58.108,160.350
C02640=1015.115,-48.575,-105.903,165.402,58.100,160.349
C02641=1015.119,-48.324,-105.914,165.405,58.093,160.349
C02642=1015.125,-48.075,-105.925,165.407,58.086,160.348
C02643=1015.129,-47.825,-105.935,165.410,58.079,160.347
C02644=1015.135,-47.576,-105.946,165.412,58.071,160.347
C02645=1015.140,-47.325,-105.957,165.415,58.064,160.346
C02646=1015.145,-47.076,-105.967,165.418,58.057,160.345
C02647=1015.150,-46.826,-105.978,165.421,58.050,160.345
C02648=1015.155,-46.576,-105.988,165.423,58.042,160.344
///RCONF 1,0,0,0,0,0,0,0,0,0,0,0,0,0,0,0,0,0,0,0,0,0,0,0
C02649=1015.159,-46.327,-105.999,165.426,58.035,160.343
C02650=1015.165,-46.077,-106.009,165.429,58.028,160.343
C02651=1015.170,-45.827,-106.021,165.431,58.020,160.342
C02652=1015.175,-45.578,-106.031,165.434,58.013,160.341
C02653=1015.180,-45.328,-106.042,165.436,58.005,160.340
C02654=1015.185,-45.078,-106.053,165.439,57.998,160.340
C02655=1015.190,-44.828,-106.063,165.443,57.990,160.340
C02656=1015.195,-44.579,-106.074,165.445,57.983,160.339
C02657=1015.201,-44.329,-106.084,165.448,57.976,160.338
C02658=1015.205,-44.080,-106.095,165.450,57.968,160.337
C02659=1015.211,-43.830,-106.106,165.453,57.961,160.337
C02660=1015.216,-43.580,-106.117,165.456,57.954,160.336
C02661=1015.221,-43.330,-106.127,165.458,57.946,160.335
C02662=1015.225,-43.081,-106.138,165.461,57.939,160.335
C02663=1015.231,-42.831,-106.149,165.463,57.931,160.334
C02664=1015.236,-42.581,-106.160,165.466,57.924,160.333
C02665=1015.242,-42.331,-106.171,165.469,57.916,160.332
C02666=1015.246,-42.081,-106.181,165.472,57.909,160.332
C02667=1015.251,-41.832,-106.192,165.474,57.901,160.331
C02668=1015.256,-41.582,-106.204,165.477,57.894,160.330
C02669=1015.262,-41.332,-106.214,165.479,57.886,160.330
C02670=1015.266,-41.083,-106.225,165.482,57.879,160.329
C02671=1015.272,-40.833,-106.236,165.484,57.871,160.328
C02672=1015.277,-40.583,-106.246,165.487,57.864,160.328
C02673=1015.282,-40.334,-106.257,165.490,57.856,160.327
C02674=1015.287,-40.083,-106.268,165.493,57.848,160.326
C02675=1015.292,-39.834,-106.279,165.495,57.841,160.325
C02676=1015.297,-39.585,-106.290,165.498,57.833,160.325
C02677=1015.303,-39.335,-106.301,165.500,57.826,160.324
C02678=1015.308,-39.085,-106.312,165.503,57.819,160.323
C02679=1015.313,-38.835,-106.323,165.506,57.812,160.323
C02680=1015.318,-38.585,-106.335,165.508,57.805,160.322
C02681=1015.323,-38.336,-106.345,165.511,57.797,160.321
C02682=1015.328,-38.061,-106.358,165.514,57.789,160.320
C02683=1015.333,-37.785,-106.370,165.517,57.780,160.320
C02684=1015.339,-37.510,-106.382,165.520,57.773,160.319
C02685=1015.345,-37.234,-106.394,165.523,57.764,160.318
C02686=1015.350,-36.984,-106.406,165.525,57.757,160.317
C02687=1015.355,-36.734,-106.417,165.528,57.750,160.317
C02688=1015.360,-36.484,-106.429,165.530,57.742,160.316
C02689=1015.366,-36.235,-106.439,165.534,57.734,160.315
C02690=1015.371,-35.985,-106.451,165.536,57.727,160.315
C02691=1015.376,-35.735,-106.462,165.539,57.719,160.314
C02692=1015.381,-35.485,-106.474,165.542,57.712,160.313
C02693=1015.386,-35.237,-106.484,165.544,57.704,160.312
C02694=1015.390,-34.986,-106.495,165.547,57.697,160.312
C02695=1015.395,-34.736,-106.507,165.549,57.689,160.311
C02696=1015.400,-34.487,-106.518,165.552,57.682,160.310
C02697=1015.406,-34.237,-106.529,165.554,57.675,160.309
C02698=1015.411,-33.987,-106.540,165.557,57.666,160.309
C02699=1015.416,-33.737,-106.552,165.560,57.659,160.308
C02700=1015.421,-33.488,-106.563,165.563,57.652,160.307
C02701=1015.427,-33.238,-106.574,165.565,57.645,160.307
C02702=1015.435,-32.836,-106.593,165.570,57.632,160.305
C02703=1015.443,-32.432,-106.610,165.574,57.620,160.304
C02704=1015.451,-32.029,-106.629,165.578,57.607,160.303
C02705=1015.459,-31.626,-106.648,165.582,57.595,160.302
C02706=1015.465,-31.376,-106.659,165.585,57.588,160.301
C02707=1015.470,-31.127,-106.670,165.587,57.580,160.300
C02708=1015.475,-30.877,-106.682,165.590,57.572,160.299
C02709=1015.480,-30.627,-106.693,165.593,57.565,160.299
C02710=1015.486,-30.377,-106.704,165.596,57.557,160.298
C02711=1015.491,-30.128,-106.716,165.598,57.549,160.297
C02712=1015.496,-29.878,-106.727,165.601,57.542,160.296
C02713=1015.501,-29.628,-106.739,165.603,57.534,160.296
C02714=1015.507,-29.379,-106.749,165.607,57.527,160.295
C02715=1015.512,-29.129,-106.761,165.609,57.519,160.294
C02716=1015.517,-28.880,-106.773,165.611,57.511,160.293
C02717=1015.522,-28.630,-106.785,165.614,57.503,160.293
C02718=1015.527,-28.380,-106.796,165.616,57.496,160.292
C02719=1015.533,-28.130,-106.807,165.620,57.488,160.291
C02720=1015.538,-27.881,-106.818,165.622,57.480,160.290
C02721=1015.543,-27.631,-106.830,165.625,57.473,160.290
C02722=1015.548,-27.381,-106.841,165.627,57.465,160.289
C02723=1015.553,-27.132,-106.854,165.630,57.458,160.288
C02724=1015.558,-26.882,-106.865,165.632,57.450,160.287
C02725=1015.563,-26.632,-106.876,165.634,57.443,160.286
C02726=1015.568,-26.383,-106.889,165.638,57.435,160.286
C02727=1015.572,-26.133,-106.901,165.641,57.427,160.285
C02728=1015.578,-25.882,-106.913,165.643,57.420,160.284
C02729=1015.583,-25.633,-106.925,165.646,57.413,160.284
C02730=1015.588,-25.384,-106.936,165.648,57.405,160.283
C02731=1015.593,-25.134,-106.948,165.650,57.397,160.282
C02732=1015.599,-24.885,-106.960,165.653,57.390,160.281
C02733=1015.604,-24.635,-106.971,165.656,57.383,160.281
C02734=1015.609,-24.385,-106.983,165.659,57.374,160.280
C02735=1015.614,-24.136,-106.995,165.661,57.367,160.279
C02736=1015.619,-23.886,-107.006,165.664,57.359,160.278
C02737=1015.624,-23.636,-107.018,165.667,57.352,160.278
C02738=1015.629,-23.387,-107.030,165.669,57.344,160.277
C02739=1015.635,-23.136,-107.042,165.671,57.337,160.276
C02740=1015.640,-22.887,-107.053,165.675,57.328,160.275
C02741=1015.645,-22.637,-107.066,165.677,57.321,160.274
C02742=1015.652,-22.265,-107.083,165.681,57.310,160.273
C02743=1015.660,-21.891,-107.101,165.685,57.298,160.272
C02744=1015.668,-21.519,-107.119,165.689,57.287,160.271
C02745=1015.675,-21.146,-107.137,165.693,57.275,160.270
C02746=1015.681,-20.896,-107.149,165.696,57.268,160.269
C02747=1015.686,-20.647,-107.160,165.698,57.260,160.268
C02748=1015.691,-20.397,-107.172,165.700,57.252,160.267
C02749=1015.697,-20.147,-107.184,165.704,57.244,160.267
C02750=1015.702,-19.897,-107.196,165.706,57.237,160.266
C02751=1015.707,-19.648,-107.208,165.708,57.229,160.265
C02752=1015.712,-19.398,-107.220,165.711,57.221,160.264
C02753=1015.717,-19.149,-107.232,165.714,57.213,160.263
C02754=1015.723,-18.898,-107.244,165.717,57.205,160.263
C02755=1015.728,-18.649,-107.256,165.719,57.198,160.262
C02756=1015.732,-18.399,-107.268,165.721,57.190,160.261
C02757=1015.738,-18.150,-107.280,165.725,57.182,160.260
C02758=1015.743,-17.900,-107.291,165.727,57.174,160.259
C02759=1015.749,-17.650,-107.304,165.729,57.166,160.258
C02760=1015.754,-17.400,-107.316,165.732,57.159,160.258
C02761=1015.759,-17.151,-107.328,165.735,57.151,160.257
C02762=1015.764,-16.902,-107.339,165.738,57.143,160.256
C02763=1015.770,-16.652,-107.352,165.740,57.135,160.255
C02764=1015.775,-16.402,-107.364,165.742,57.128,160.254
C02765=1015.780,-16.153,-107.375,165.746,57.119,160.254
C02766=1015.785,-15.903,-107.388,165.748,57.112,160.253
C02767=1015.790,-15.653,-107.400,165.750,57.104,160.252
C02768=1015.796,-15.403,-107.412,165.753,57.096,160.251
C02769=1015.800,-15.154,-107.425,165.755,57.089,160.250
C02770=1015.806,-14.904,-107.438,165.758,57.081,160.249
C02771=1015.811,-14.654,-107.449,165.762,57.074,160.249
C02772=1015.816,-14.405,-107.462,165.764,57.066,160.248
C02773=1015.822,-14.155,-107.474,165.766,57.058,160.247
C02774=1015.826,-13.905,-107.486,165.769,57.051,160.246
C02775=1015.831,-13.656,-107.499,165.771,57.043,160.245
C02776=1015.836,-13.406,-107.511,165.774,57.035,160.245
C02777=1015.842,-13.156,-107.524,165.777,57.027,160.244
C02778=1015.847,-12.907,-107.536,165.779,57.019,160.243
C02779=1015.852,-12.657,-107.548,165.782,57.012,160.242
C02780=1015.857,-12.407,-107.561,165.784,57.004,160.241
C02781=1015.862,-12.158,-107.573,165.786,56.996,160.241
C02782=1015.868,-11.909,-107.585,165.790,56.988,160.240
C02783=1015.873,-11.658,-107.598,165.792,56.981,160.239
C02784=1015.878,-11.409,-107.610,165.795,56.973,160.238
C02785=1015.883,-11.160,-107.622,165.797,56.965,160.237
C02786=1015.888,-10.909,-107.635,165.800,56.957,160.237
C02787=1015.894,-10.660,-107.647,165.803,56.950,160.236
C02788=1015.898,-10.411,-107.660,165.805,56.942,160.235
C02789=1015.904,-10.161,-107.673,165.808,56.934,160.234
C02790=1015.909,-9.911,-107.684,165.810,56.927,160.233
C02791=1015.914,-9.661,-107.697,165.814,56.919,160.233
C02792=1015.920,-9.412,-107.709,165.816,56.911,160.232
C02793=1015.925,-9.162,-107.722,165.818,56.902,160.231
C02794=1015.930,-8.912,-107.735,165.820,56.895,160.230
C02795=1015.935,-8.663,-107.747,165.824,56.887,160.229
C02796=1015.940,-8.414,-107.760,165.826,56.879,160.228
C02797=1015.946,-8.164,-107.772,165.828,56.871,160.227
C02798=1015.951,-7.914,-107.784,165.831,56.864,160.226
C02799=1015.956,-7.664,-107.797,165.834,56.856,160.226
C02800=1015.961,-7.414,-107.809,165.837,56.848,160.225
C02801=1015.967,-7.165,-107.821,165.839,56.840,160.224
C02802=1015.972,-6.915,-107.834,165.842,56.832,160.223
C02803=1015.977,-6.666,-107.847,165.844,56.824,160.222
C02804=1015.983,-6.416,-107.859,165.847,56.816,160.221
C02805=1015.988,-6.167,-107.872,165.849,56.809,160.221
C02806=1015.993,-5.888,-107.886,165.852,56.800,160.220
C02807=1015.999,-5.609,-107.900,165.855,56.790,160.218
C02808=1016.006,-5.331,-107.913,165.857,56.781,160.217
C02809=1016.012,-5.054,-107.928,165.860,56.773,160.216
C02810=1016.017,-4.803,-107.941,165.864,56.765,160.216
C02811=1016.022,-4.554,-107.953,165.866,56.757,160.215
C02812=1016.027,-4.304,-107.966,165.869,56.749,160.214
C02813=1016.032,-4.055,-107.979,165.871,56.742,160.213
C02814=1016.038,-3.805,-107.992,165.875,56.734,160.213
C02815=1016.042,-3.555,-108.004,165.877,56.726,160.212
C02816=1016.047,-3.305,-108.018,165.880,56.718,160.211
C02817=1016.053,-3.056,-108.031,165.882,56.711,160.210
C02818=1016.058,-2.806,-108.044,165.884,56.703,160.209
C02819=1016.063,-2.557,-108.056,165.887,56.695,160.208
C02820=1016.068,-2.306,-108.070,165.889,56.688,160.207
C02821=1016.073,-2.057,-108.082,165.892,56.679,160.206
C02822=1016.079,-1.808,-108.096,165.895,56.671,160.206
C02823=1016.083,-1.558,-108.108,165.897,56.664,160.205
C02824=1016.088,-1.308,-108.122,165.900,56.656,160.204
C02825=1016.094,-1.059,-108.134,165.902,56.649,160.203
C02826=1016.099,-0.809,-108.148,165.904,56.641,160.202
C02827=1016.104,-0.560,-108.160,165.908,56.633,160.202
C02828=1016.109,-0.310,-108.174,165.910,56.625,160.201
C02829=1016.115,-0.061,-108.186,165.913,56.618,160.200
C02830=1016.120,0.189,-108.200,165.915,56.610,160.199
C02831=1016.124,0.439,-108.212,165.917,56.602,160.198
C02832=1016.130,0.688,-108.226,165.920,56.594,160.197
C02833=1016.135,0.937,-108.238,165.923,56.586,160.196
C02834=1016.140,1.188,-108.252,165.926,56.578,160.196
C02835=1016.145,1.438,-108.265,165.928,56.571,160.195
C02836=1016.150,1.687,-108.278,165.931,56.563,160.194
C02837=1016.156,1.937,-108.291,165.932,56.555,160.193
C02838=1016.161,2.186,-108.304,165.936,56.547,160.192
C02839=1016.166,2.436,-108.317,165.938,56.539,160.191
C02840=1016.171,2.685,-108.330,165.941,56.532,160.190
C02841=1016.177,2.934,-108.343,165.943,56.524,160.189
C02842=1016.182,3.185,-108.357,165.946,56.515,160.189
C02843=1016.187,3.434,-108.369,165.949,56.508,160.188
C02844=1016.192,3.684,-108.383,165.951,56.500,160.187
C02845=1016.198,3.933,-108.395,165.954,56.492,160.186
C02846=1016.203,4.183,-108.409,165.957,56.484,160.185
C02847=1016.208,4.433,-108.422,165.959,56.476,160.184
C02848=1016.213,4.682,-108.435,165.962,56.468,160.183
C02849=1016.219,4.931,-108.449,165.964,56.460,160.182
C02850=1016.224,5.181,-108.461,165.967,56.452,160.182
C02851=1016.229,5.431,-108.474,165.970,56.444,160.181
C02852=1016.234,5.681,-108.488,165.972,56.436,160.180
C02853=1016.239,5.930,-108.501,165.974,56.428,160.179
C02854=1016.245,6.179,-108.514,165.978,56.420,160.178
C02855=1016.250,6.430,-108.528,165.980,56.412,160.177
C02856=1016.255,6.678,-108.541,165.982,56.405,160.176
C02857=1016.260,6.929,-108.554,165.984,56.397,160.175
C02858=1016.266,7.178,-108.567,165.987,56.388,160.174
C02859=1016.271,7.427,-108.580,165.990,56.381,160.173
C02860=1016.276,7.677,-108.594,165.992,56.373,160.173
C02861=1016.282,7.927,-108.607,165.995,56.364,160.172
C02862=1016.287,8.176,-108.619,165.998,56.357,160.171
C02863=1016.292,8.426,-108.633,166.000,56.348,160.170
C02864=1016.298,8.676,-108.646,166.002,56.341,160.169
C02865=1016.302,8.925,-108.660,166.006,56.333,160.168
C02866=1016.308,9.175,-108.672,166.008,56.324,160.167
C02867=1016.314,9.424,-108.686,166.010,56.317,160.166
C02868=1016.319,9.673,-108.700,166.013,56.308,160.165
C02869=1016.324,9.924,-108.713,166.016,56.301,160.164
C02870=1016.330,10.204,-108.728,166.018,56.291,160.163
C02871=1016.336,10.484,-108.743,166.021,56.282,160.162
C02872=1016.342,10.765,-108.758,166.024,56.274,160.161
C02873=1016.348,11.046,-108.773,166.027,56.264,160.160
C02874=1016.353,11.295,-108.787,166.030,56.256,160.159
C02875=1016.359,11.544,-108.799,166.032,56.248,160.158
C02876=1016.364,11.794,-108.813,166.035,56.240,160.157
C02877=1016.369,12.044,-108.826,166.038,56.232,160.157
C02878=1016.375,12.294,-108.840,166.040,56.224,160.156
C02879=1016.381,12.542,-108.853,166.042,56.216,160.155
C02880=1016.386,12.793,-108.866,166.046,56.207,160.154
C02881=1016.391,13.042,-108.880,166.048,56.199,160.153
C02882=1016.397,13.292,-108.893,166.050,56.191,160.152
C02883=1016.402,13.542,-108.907,166.054,56.183,160.151
C02884=1016.407,13.791,-108.920,166.056,56.176,160.150
C02885=1016.412,14.040,-108.934,166.058,56.167,160.149
C02886=1016.417,14.291,-108.947,166.061,56.160,160.148
C02887=1016.423,14.540,-108.961,166.063,56.152,160.147
C02888=1016.428,14.790,-108.975,166.066,56.143,160.146
C02889=1016.432,15.039,-108.989,166.069,56.136,160.146
C02890=1016.438,15.288,-109.003,166.071,56.128,160.144
C02891=1016.443,15.539,-109.016,166.073,56.120,160.144
C02892=1016.449,15.788,-109.030,166.077,56.112,160.143
C02893=1016.454,16.038,-109.044,166.079,56.104,160.142
C02894=1016.459,16.287,-109.057,166.081,56.096,160.141
C02895=1016.464,16.536,-109.071,166.083,56.088,160.140
C02896=1016.470,16.786,-109.084,166.087,56.080,160.139
C02897=1016.475,17.036,-109.098,166.089,56.072,160.138
C02898=1016.480,17.286,-109.112,166.092,56.064,160.137
C02899=1016.485,17.534,-109.125,166.094,56.056,160.136
C02900=1016.491,17.784,-109.139,166.097,56.048,160.136
C02901=1016.496,18.034,-109.153,166.099,56.040,160.134
C02902=1016.502,18.283,-109.167,166.102,56.032,160.134
C02903=1016.507,18.533,-109.181,166.104,56.024,160.132
C02904=1016.512,18.783,-109.195,166.107,56.016,160.132
C02905=1016.517,19.032,-109.208,166.109,56.008,160.131
C02906=1016.522,19.282,-109.222,166.112,56.000,160.130
C02907=1016.528,19.531,-109.236,166.114,55.992,160.129
C02908=1016.533,19.781,-109.250,166.118,55.984,160.128
C02909=1016.538,20.031,-109.264,166.120,55.976,160.127
C02910=1016.543,20.280,-109.278,166.122,55.968,160.126
C02911=1016.549,20.530,-109.292,166.125,55.960,160.125
C02912=1016.554,20.779,-109.306,166.128,55.952,160.124
C02913=1016.559,21.028,-109.319,166.130,55.944,160.124
C02914=1016.564,21.278,-109.334,166.132,55.936,160.122
C02915=1016.569,21.528,-109.348,166.135,55.928,160.122
C02916=1016.575,21.777,-109.361,166.137,55.920,160.120
C02917=1016.580,22.027,-109.375,166.141,55.912,160.120
C02918=1016.585,22.277,-109.390,166.143,55.904,160.119
C02919=1016.590,22.526,-109.404,166.145,55.896,160.118
C02920=1016.596,22.776,-109.417,166.147,55.888,160.117
C02921=1016.601,23.026,-109.431,166.151,55.880,160.116
C02922=1016.607,23.274,-109.446,166.153,55.872,160.115
C02923=1016.611,23.524,-109.460,166.155,55.864,160.114
C02924=1016.617,23.773,-109.474,166.157,55.856,160.113
C02925=1016.622,24.023,-109.488,166.161,55.848,160.112
C02926=1016.628,24.272,-109.502,166.163,55.840,160.111
C02927=1016.632,24.522,-109.516,166.165,55.832,160.110
C02928=1016.638,24.772,-109.530,166.169,55.824,160.109
C02929=1016.643,25.021,-109.544,166.171,55.816,160.108
C02930=1016.649,25.271,-109.558,166.174,55.808,160.108
C02931=1016.654,25.521,-109.572,166.176,55.800,160.106
C02932=1016.659,25.770,-109.587,166.179,55.791,160.106
C02933=1016.665,26.019,-109.601,166.181,55.784,160.105
C02934=1016.671,26.301,-109.616,166.184,55.774,160.103
C02935=1016.677,26.584,-109.632,166.187,55.766,160.103
C02936=1016.682,26.865,-109.649,166.190,55.756,160.101
C02937=1016.689,27.148,-109.665,166.192,55.747,160.100
C02938=1016.693,27.397,-109.678,166.196,55.739,160.099
C02939=1016.700,27.647,-109.693,166.198,55.731,160.098
C02940=1016.705,27.896,-109.708,166.200,55.723,160.098
C02941=1016.710,28.146,-109.721,166.203,55.715,160.096
C02942=1016.715,28.396,-109.736,166.205,55.707,160.096
C02943=1016.721,28.645,-109.750,166.207,55.699,160.095
C02944=1016.725,28.895,-109.765,166.211,55.691,160.094
C02945=1016.731,29.144,-109.779,166.213,55.683,160.093
C02946=1016.736,29.394,-109.794,166.216,55.676,160.092
C02947=1016.741,29.643,-109.808,166.218,55.667,160.091
C02948=1016.746,29.893,-109.822,166.221,55.659,160.090
C02949=1016.752,30.142,-109.837,166.223,55.651,160.089
C02950=1016.757,30.392,-109.851,166.226,55.643,160.088
C02951=1016.762,30.641,-109.865,166.228,55.636,160.087
C02952=1016.767,30.891,-109.880,166.230,55.627,160.086
C02953=1016.773,31.140,-109.894,166.234,55.619,160.085
C02954=1016.777,31.390,-109.909,166.236,55.611,160.084
C02955=1016.783,31.639,-109.923,166.239,55.604,160.083
C02956=1016.788,31.889,-109.938,166.241,55.595,160.082
C02957=1016.794,32.138,-109.952,166.244,55.587,160.081
C02958=1016.798,32.388,-109.967,166.246,55.579,160.081
C02959=1016.804,32.637,-109.981,166.249,55.571,160.079
C02960=1016.809,32.887,-109.996,166.251,55.563,160.078
C02961=1016.814,33.136,-110.010,166.254,55.555,160.078
C02962=1016.820,33.385,-110.024,166.256,55.547,160.077
C02963=1016.825,33.635,-110.039,166.259,55.539,160.076
C02964=1016.830,33.885,-110.053,166.261,55.531,160.075
C02965=1016.836,34.135,-110.068,166.264,55.523,160.074
C02966=1016.841,34.384,-110.082,166.266,55.514,160.073
C02967=1016.846,34.634,-110.097,166.269,55.507,160.072
C02968=1016.852,34.883,-110.111,166.272,55.498,160.071
C02969=1016.857,35.132,-110.126,166.274,55.490,160.070
C02970=1016.862,35.382,-110.140,166.277,55.483,160.069
C02971=1016.868,35.631,-110.155,166.279,55.474,160.068
C02972=1016.873,35.881,-110.169,166.282,55.466,160.067
C02973=1016.878,36.130,-110.184,166.284,55.458,160.066
C02974=1016.884,36.380,-110.199,166.287,55.450,160.065
C02975=1016.889,36.630,-110.214,166.289,55.442,160.064
C02976=1016.894,36.879,-110.228,166.292,55.433,160.063
C02977=1016.899,37.129,-110.243,166.295,55.426,160.062
C02978=1016.904,37.378,-110.257,166.297,55.418,160.061
C02979=1016.909,37.628,-110.272,166.300,55.410,160.060
C02980=1016.914,37.877,-110.288,166.302,55.402,160.059
C02981=1016.920,38.127,-110.302,166.305,55.393,160.058
C02982=1016.926,38.376,-110.317,166.308,55.386,160.057
C02983=1016.931,38.626,-110.332,166.310,55.378,160.056
C02984=1016.935,38.876,-110.347,166.313,55.370,160.056
C02985=1016.941,39.124,-110.361,166.315,55.362,160.054
C02986=1016.946,39.374,-110.376,166.318,55.353,160.054
C02987=1016.952,39.624,-110.391,166.321,55.346,160.053
C02988=1016.957,39.874,-110.406,166.323,55.338,160.052
C02989=1016.962,40.123,-110.421,166.325,55.330,160.051
C02990=1016.967,40.372,-110.435,166.328,55.322,160.050
C02991=1016.972,40.622,-110.451,166.331,55.314,160.049
C02992=1016.977,40.871,-110.466,166.333,55.305,160.048
C02993=1016.983,41.121,-110.480,166.336,55.298,160.047
C02994=1016.988,41.371,-110.495,166.338,55.290,160.046
C02995=1016.993,41.620,-110.510,166.341,55.281,160.045
C02996=1016.998,41.869,-110.525,166.344,55.274,160.044
C02997=1017.004,42.119,-110.539,166.346,55.266,160.043
C02998=1017.010,42.401,-110.557,166.349,55.256,160.042
C02999=1017.015,42.683,-110.574,166.352,55.248,160.041
C03000=1017.022,42.965,-110.592,166.355,55.238,160.040
C03001=1017.028,43.247,-110.609,166.358,55.230,160.039
C03002=1017.033,43.496,-110.624,166.360,55.222,160.038
C03003=1017.038,43.746,-110.638,166.363,55.214,160.037
C03004=1017.043,43.996,-110.654,166.365,55.206,160.036
C03005=1017.048,44.245,-110.669,166.367,55.198,160.035
C03006=1017.053,44.495,-110.684,166.370,55.190,160.034
C03007=1017.058,44.744,-110.700,166.373,55.182,160.033
C03008=1017.063,44.993,-110.715,166.376,55.174,160.032
C03009=1017.068,45.243,-110.731,166.378,55.166,160.031
C03010=1017.073,45.493,-110.746,166.380,55.159,160.030
C03011=1017.078,45.742,-110.761,166.383,55.151,160.029
C03012=1017.083,45.991,-110.776,166.385,55.143,160.028
C03013=1017.088,46.241,-110.792,166.388,55.135,160.027
C03014=1017.094,46.491,-110.807,166.391,55.127,160.026
C03015=1017.099,46.740,-110.822,166.393,55.118,160.025
C03016=1017.104,46.989,-110.837,166.396,55.111,160.024
C03017=1017.109,47.238,-110.853,166.398,55.103,160.023
C03018=1017.115,47.488,-110.868,166.400,55.095,160.022
C03019=1017.120,47.738,-110.883,166.403,55.087,160.021
C03020=1017.125,47.987,-110.899,166.406,55.079,160.020
C03021=1017.131,48.237,-110.914,166.409,55.071,160.020
C03022=1017.136,48.486,-110.929,166.411,55.063,160.019
C03023=1017.141,48.735,-110.944,166.413,55.055,160.018
C03024=1017.146,48.985,-110.960,166.415,55.047,160.016
C03025=1017.151,49.235,-110.975,166.418,55.039,160.016
C03026=1017.156,49.484,-110.990,166.421,55.031,160.015
C03027=1017.161,49.733,-111.005,166.424,55.023,160.014
C03028=1017.167,49.983,-111.021,166.426,55.015,160.013
C03029=1017.172,50.232,-111.036,166.428,55.007,160.012
C03030=1017.177,50.482,-111.051,166.431,54.999,160.011
C03031=1017.183,50.732,-111.067,166.434,54.991,160.010
C03032=1017.188,50.981,-111.082,166.437,54.983,160.009
C03033=1017.193,51.230,-111.099,166.439,54.975,160.008
C03034=1017.198,51.480,-111.114,166.441,54.967,160.007
C03035=1017.203,51.729,-111.129,166.444,54.958,160.006
C03036=1017.208,51.978,-111.144,166.447,54.951,160.005
C03037=1017.214,52.228,-111.160,166.449,54.943,160.004
C03038=1017.219,52.478,-111.175,166.452,54.935,160.003
C03039=1017.224,52.727,-111.190,166.454,54.927,160.002
C03040=1017.230,52.977,-111.206,166.457,54.918,160.001
C03041=1017.235,53.226,-111.221,166.460,54.911,160.000
C03042=1017.241,53.475,-111.237,166.462,54.903,159.999
C03043=1017.246,53.725,-111.252,166.464,54.894,159.998
C03044=1017.251,53.974,-111.268,166.468,54.886,159.997
C03045=1017.256,54.224,-111.283,166.470,54.878,159.996
C03046=1017.261,54.473,-111.298,166.473,54.870,159.995
C03047=1017.267,54.723,-111.314,166.475,54.862,159.994
C03048=1017.272,54.972,-111.329,166.478,54.854,159.993
C03049=1017.277,55.221,-111.345,166.480,54.846,159.992
C03050=1017.283,55.471,-111.361,166.483,54.838,159.991
C03051=1017.288,55.720,-111.376,166.485,54.829,159.990
C03052=1017.293,55.971,-111.392,166.488,54.821,159.989
C03053=1017.298,56.220,-111.407,166.491,54.814,159.988
C03054=1017.303,56.469,-111.423,166.493,54.805,159.987
C03055=1017.309,56.719,-111.438,166.495,54.797,159.986
C03056=1017.314,56.968,-111.454,166.499,54.789,159.985
C03057=1017.320,57.218,-111.469,166.501,54.781,159.984
C03058=1017.325,57.467,-111.484,166.503,54.773,159.983
C03059=1017.331,57.716,-111.501,166.505,54.764,159.982
C03060=1017.336,57.966,-111.516,166.509,54.756,159.981
C03061=1017.341,58.216,-111.531,166.511,54.748,159.980
C03062=1017.347,58.497,-111.549,166.514,54.739,159.979
C03063=1017.353,58.779,-111.566,166.517,54.729,159.978
C03064=1017.360,59.061,-111.584,166.519,54.720,159.976
C03065=1017.366,59.343,-111.602,166.522,54.711,159.975
C03066=1017.371,59.593,-111.617,166.526,54.703,159.974
C03067=1017.377,59.842,-111.633,166.528,54.694,159.973
C03068=1017.382,60.091,-111.648,166.531,54.687,159.972
C03069=1017.387,60.341,-111.664,166.534,54.679,159.972
C03070=1017.393,60.590,-111.680,166.536,54.671,159.970
C03071=1017.398,60.840,-111.696,166.539,54.662,159.969
C03072=1017.403,61.089,-111.711,166.542,54.654,159.968
C03073=1017.409,61.339,-111.727,166.544,54.646,159.967
C03074=1017.414,61.588,-111.742,166.546,54.638,159.966
C03075=1017.419,61.838,-111.758,166.550,54.629,159.965
C03076=1017.424,62.087,-111.773,166.552,54.621,159.964
C03077=1017.430,62.337,-111.789,166.554,54.613,159.963
C03078=1017.435,62.586,-111.804,166.557,54.604,159.962
C03079=1017.441,62.835,-111.821,166.560,54.597,159.961
C03080=1017.446,63.085,-111.837,166.562,54.589,159.960
C03081=1017.451,63.335,-111.852,166.565,54.580,159.959
C03082=1017.457,63.583,-111.868,166.567,54.572,159.958
C03083=1017.461,63.834,-111.884,166.570,54.564,159.957
C03084=1017.467,64.082,-111.900,166.573,54.556,159.956
C03085=1017.472,64.332,-111.917,166.575,54.548,159.955
C03086=1017.478,64.582,-111.932,166.578,54.540,159.954
C03087=1017.483,64.831,-111.948,166.581,54.532,159.953
C03088=1017.488,65.081,-111.964,166.583,54.524,159.952
C03089=1017.493,65.330,-111.980,166.586,54.516,159.951
C03090=1017.499,65.580,-111.996,166.588,54.508,159.950
C03091=1017.504,65.829,-112.012,166.590,54.500,159.949
C03092=1017.509,66.079,-112.028,166.594,54.491,159.948
C03093=1017.514,66.327,-112.044,166.596,54.484,159.947
C03094=1017.520,66.577,-112.061,166.599,54.476,159.946
C03095=1017.525,66.827,-112.077,166.601,54.468,159.945
C03096=1017.530,67.076,-112.093,166.604,54.459,159.944
C03097=1017.536,67.326,-112.108,166.607,54.451,159.943
C03098=1017.540,67.575,-112.125,166.609,54.443,159.942
C03099=1017.546,67.824,-112.141,166.611,54.435,159.941
C03100=1017.551,68.074,-112.157,166.614,54.427,159.940
C03101=1017.556,68.323,-112.173,166.618,54.419,159.939
C03102=1017.562,68.573,-112.190,166.620,54.411,159.938
C03103=1017.567,68.822,-112.205,166.622,54.403,159.937
C03104=1017.572,69.072,-112.222,166.625,54.395,159.936
C03105=1017.577,69.321,-112.239,166.627,54.387,159.935
C03106=1017.582,69.570,-112.255,166.630,54.379,159.934
C03107=1017.587,69.820,-112.271,166.633,54.371,159.934
C03108=1017.593,70.069,-112.287,166.635,54.363,159.932
C03109=1017.598,70.318,-112.303,166.638,54.355,159.931
C03110=1017.604,70.568,-112.320,166.640,54.347,159.930
C03111=1017.608,70.817,-112.335,166.644,54.339,159.929
C03112=1017.613,71.067,-112.352,166.646,54.331,159.928
C03113=1017.619,71.316,-112.369,166.648,54.323,159.927
C03114=1017.624,71.565,-112.385,166.651,54.315,159.926
C03115=1017.629,71.815,-112.402,166.653,54.307,159.925
C03116=1017.634,72.064,-112.417,166.657,54.299,159.925
C03117=1017.639,72.314,-112.434,166.659,54.291,159.923
C03118=1017.645,72.563,-112.450,166.662,54.283,159.922
C03119=1017.650,72.812,-112.467,166.664,54.275,159.921
C03120=1017.655,73.062,-112.483,166.666,54.267,159.920
C03121=1017.661,73.311,-112.500,166.670,54.258,159.919
C03122=1017.665,73.561,-112.516,166.672,54.250,159.918
C03123=1017.671,73.810,-112.532,166.675,54.243,159.918
C03124=1017.677,74.060,-112.549,166.677,54.235,159.916
C03125=1017.681,74.309,-112.565,166.680,54.227,159.915
C03126=1017.688,74.591,-112.583,166.684,54.217,159.914
C03127=1017.693,74.873,-112.602,166.687,54.208,159.913
C03128=1017.700,75.155,-112.621,166.689,54.199,159.912
C03129=1017.706,75.437,-112.639,166.692,54.190,159.911
C03130=1017.711,75.686,-112.656,166.695,54.182,159.910
C03131=1017.716,75.935,-112.673,166.697,54.174,159.909
C03132=1017.721,76.185,-112.690,166.700,54.166,159.908
C03133=1017.726,76.434,-112.705,166.703,54.158,159.907
C03134=1017.731,76.684,-112.722,166.705,54.150,159.906
C03135=1017.737,76.934,-112.738,166.708,54.142,159.905
C03136=1017.742,77.183,-112.755,166.710,54.134,159.904
C03137=1017.747,77.432,-112.771,166.713,54.126,159.903
C03138=1017.753,77.681,-112.789,166.715,54.118,159.902
C03139=1017.758,77.931,-112.806,166.719,54.110,159.901
C03140=1017.763,78.180,-112.822,166.721,54.102,159.900
C03141=1017.768,78.429,-112.839,166.724,54.094,159.899
C03142=1017.773,78.679,-112.856,166.726,54.087,159.898
C03143=1017.778,78.929,-112.873,166.729,54.079,159.897
C03144=1017.783,79.178,-112.889,166.731,54.071,159.896
C03145=1017.788,79.427,-112.906,166.735,54.062,159.895
C03146=1017.793,79.677,-112.923,166.737,54.054,159.894
C03147=1017.798,79.927,-112.940,166.739,54.046,159.893
C03148=1017.804,80.175,-112.956,166.742,54.039,159.892
C03149=1017.809,80.424,-112.973,166.745,54.031,159.891
C03150=1017.814,80.674,-112.990,166.747,54.023,159.890
C03151=1017.820,80.924,-113.007,166.751,54.015,159.889
C03152=1017.824,81.172,-113.023,166.753,54.007,159.888
C03153=1017.830,81.422,-113.040,166.755,53.999,159.887
C03154=1017.835,81.671,-113.058,166.758,53.991,159.886
C03155=1017.840,81.921,-113.075,166.760,53.983,159.885
C03156=1017.845,82.170,-113.091,166.764,53.974,159.884
C03157=1017.850,82.419,-113.108,166.767,53.967,159.883
C03158=1017.855,82.669,-113.125,166.769,53.959,159.882
C03159=1017.861,82.919,-113.142,166.771,53.951,159.881
C03160=1017.867,83.167,-113.159,166.774,53.943,159.880
C03161=1017.872,83.417,-113.175,166.777,53.935,159.879
C03162=1017.877,83.666,-113.192,166.780,53.927,159.878
C03163=1017.882,83.916,-113.209,166.782,53.919,159.877
C03164=1017.887,84.165,-113.226,166.785,53.911,159.876
C03165=1017.893,84.414,-113.243,166.787,53.903,159.875
C03166=1017.898,84.664,-113.260,166.791,53.894,159.874
C03167=1017.903,84.914,-113.277,166.793,53.886,159.873
C03168=1017.908,85.163,-113.293,166.795,53.878,159.872
C03169=1017.913,85.412,-113.311,166.798,53.870,159.871
C03170=1017.918,85.661,-113.328,166.801,53.862,159.870
C03171=1017.924,85.911,-113.345,166.804,53.854,159.869
C03172=1017.929,86.161,-113.362,166.806,53.846,159.868
C03173=1017.934,86.410,-113.379,166.809,53.838,159.867
C03174=1017.940,86.658,-113.395,166.812,53.830,159.866
C03175=1017.945,86.908,-113.412,166.815,53.822,159.865
C03176=1017.950,87.157,-113.429,166.817,53.814,159.864
C03177=1017.956,87.407,-113.446,166.819,53.806,159.863
C03178=1017.961,87.656,-113.463,166.823,53.797,159.862
C03179=1017.966,87.906,-113.481,166.825,53.789,159.861
C03180=1017.971,88.155,-113.498,166.828,53.782,159.860
C03181=1017.977,88.405,-113.514,166.830,53.774,159.859
C03182=1017.982,88.655,-113.531,166.834,53.765,159.858
C03183=1017.987,88.903,-113.548,166.836,53.757,159.857
C03184=1017.992,89.152,-113.565,166.839,53.749,159.856
C03185=1017.998,89.402,-113.583,166.842,53.742,159.855
C03186=1018.002,89.652,-113.600,166.844,53.734,159.854
C03187=1018.008,89.901,-113.618,166.848,53.726,159.853
C03188=1018.013,90.150,-113.635,166.850,53.718,159.852
C03189=1018.018,90.399,-113.652,166.853,53.710,159.851
C03190=1018.023,90.681,-113.672,166.856,53.701,159.850
C03191=1018.030,90.964,-113.691,166.859,53.692,159.849
C03192=1018.035,91.246,-113.711,166.862,53.683,159.848
C03193=1018.041,91.527,-113.730,166.865,53.674,159.847
C03194=1018.046,91.776,-113.748,166.868,53.666,159.846
C03195=1018.052,92.026,-113.765,166.870,53.659,159.845
C03196=1018.056,92.275,-113.783,166.873,53.651,159.844
C03197=1018.062,92.525,-113.800,166.876,53.642,159.843
C03198=1018.067,92.774,-113.817,166.879,53.634,159.842
C03199=1018.072,93.024,-113.834,166.881,53.626,159.841
C03200=1018.077,93.273,-113.852,166.884,53.618,159.840
C03201=1018.083,93.522,-113.870,166.886,53.611,159.839
C03202=1018.088,93.772,-113.887,166.890,53.602,159.838
C03203=1018.093,94.021,-113.904,166.893,53.595,159.837
C03204=1018.098,94.271,-113.922,166.895,53.587,159.836
C03205=1018.103,94.520,-113.939,166.898,53.579,159.835
C03206=1018.109,94.769,-113.957,166.900,53.571,159.834
C03207=1018.114,95.018,-113.974,166.904,53.563,159.833
C03208=1018.119,95.268,-113.992,166.906,53.555,159.832
C03209=1018.124,95.517,-114.010,166.909,53.547,159.831
C03210=1018.130,95.767,-114.026,166.911,53.539,159.830
C03211=1018.135,96.016,-114.044,166.915,53.531,159.829
C03212=1018.140,96.266,-114.061,166.917,53.523,159.828
C03213=1018.145,96.515,-114.079,166.920,53.515,159.827
C03214=1018.151,96.764,-114.097,166.922,53.507,159.826
C03215=1018.156,97.013,-114.113,166.926,53.499,159.825
C03216=1018.161,97.263,-114.132,166.928,53.491,159.824
C03217=1018.166,97.512,-114.149,166.931,53.483,159.823
C03218=1018.172,97.761,-114.167,166.933,53.475,159.822
C03219=1018.177,98.010,-114.184,166.937,53.467,159.821
C03220=1018.182,98.260,-114.202,166.939,53.459,159.820
C03221=1018.187,98.509,-114.219,166.942,53.451,159.819
C03222=1018.192,98.758,-114.236,166.944,53.443,159.818
C03223=1018.198,99.007,-114.254,166.948,53.435,159.817
C03224=1018.203,99.257,-114.272,166.950,53.427,159.816
C03225=1018.208,99.506,-114.289,166.953,53.419,159.815
C03226=1018.213,99.756,-114.307,166.955,53.411,159.814
C03227=1018.217,100.005,-114.325,166.958,53.403,159.813
C03228=1018.223,100.254,-114.343,166.961,53.396,159.812
C03229=1018.228,100.504,-114.361,166.964,53.387,159.811
C03230=1018.233,100.753,-114.378,166.967,53.380,159.810
C03231=1018.238,101.002,-114.397,166.970,53.372,159.809
C03232=1018.243,101.251,-114.414,166.972,53.364,159.808
C03233=1018.248,101.500,-114.432,166.975,53.356,159.807
C03234=1018.254,101.749,-114.450,166.978,53.348,159.806
C03235=1018.259,101.999,-114.468,166.981,53.340,159.805
C03236=1018.264,102.249,-114.486,166.984,53.333,159.804
C03237=1018.269,102.498,-114.503,166.986,53.325,159.803
C03238=1018.274,102.748,-114.522,166.989,53.317,159.802
C03239=1018.279,102.997,-114.539,166.992,53.308,159.801
C03240=1018.284,103.246,-114.557,166.995,53.301,159.800
C03241=1018.290,103.495,-114.575,166.997,53.293,159.799
C03242=1018.295,103.745,-114.593,167.000,53.285,159.798
C03243=1018.300,103.994,-114.611,167.003,53.277,159.797
C03244=1018.305,104.243,-114.629,167.006,53.269,159.796
C03245=1018.310,104.492,-114.646,167.009,53.261,159.795
C03246=1018.316,104.742,-114.665,167.011,53.253,159.794
C03247=1018.321,104.991,-114.683,167.014,53.246,159.793
C03248=1018.326,105.240,-114.701,167.018,53.237,159.792
C03249=1018.331,105.490,-114.719,167.020,53.230,159.791
C03250=1018.336,105.739,-114.736,167.023,53.222,159.790
C03251=1018.341,105.988,-114.754,167.026,53.214,159.789
C03252=1018.347,106.237,-114.772,167.028,53.206,159.788
C03253=1018.352,106.487,-114.791,167.032,53.198,159.787
C03254=1018.357,106.769,-114.810,167.035,53.189,159.786
C03255=1018.363,107.051,-114.831,167.038,53.180,159.785
C03256=1018.369,107.334,-114.852,167.041,53.171,159.784
C03257=1018.376,107.616,-114.871,167.044,53.162,159.783
C03258=1018.381,107.865,-114.890,167.047,53.154,159.782
C03259=1018.386,108.114,-114.908,167.050,53.146,159.781
C03260=1018.391,108.363,-114.926,167.053,53.138,159.780
C03261=1018.396,108.613,-114.945,167.056,53.130,159.779
C03262=1018.402,108.862,-114.962,167.058,53.122,159.778
C03263=1018.407,109.111,-114.980,167.062,53.114,159.777
C03264=1018.412,109.360,-114.998,167.064,53.106,159.776
C03265=1018.417,109.610,-115.016,167.067,53.098,159.775
C03266=1018.422,109.860,-115.035,167.070,53.090,159.774
C03267=1018.427,110.109,-115.053,167.073,53.082,159.773
C03268=1018.433,110.358,-115.071,167.076,53.074,159.772
C03269=1018.438,110.607,-115.089,167.078,53.066,159.771
C03270=1018.443,110.856,-115.107,167.081,53.059,159.770
C03271=1018.448,111.106,-115.126,167.085,53.050,159.769
C03272=1018.454,111.355,-115.144,167.087,53.042,159.768
C03273=1018.459,111.604,-115.162,167.090,53.035,159.767
C03274=1018.463,111.853,-115.180,167.092,53.027,159.766
C03275=1018.468,112.103,-115.199,167.096,53.019,159.765
C03276=1018.474,112.352,-115.217,167.099,53.011,159.764
C03277=1018.479,112.602,-115.236,167.102,53.004,159.763
C03278=1018.483,112.851,-115.254,167.104,52.996,159.762
C03279=1018.488,113.100,-115.273,167.107,52.988,159.761
C03280=1018.494,113.350,-115.292,167.110,52.981,159.760
C03281=1018.499,113.598,-115.310,167.114,52.972,159.759
C03282=1018.504,113.848,-115.329,167.116,52.965,159.758
C03283=1018.509,114.097,-115.347,167.119,52.957,159.757
C03284=1018.514,114.346,-115.366,167.121,52.949,159.756
C03285=1018.519,114.596,-115.384,167.124,52.942,159.756
C03286=1018.524,114.845,-115.403,167.127,52.934,159.755
C03287=1018.529,115.094,-115.421,167.131,52.926,159.754
C03288=1018.534,115.343,-115.440,167.133,52.918,159.753
C03289=1018.539,115.593,-115.459,167.136,52.910,159.752
C03290=1018.544,115.842,-115.477,167.139,52.903,159.751
C03291=1018.549,116.091,-115.496,167.142,52.895,159.750
C03292=1018.555,116.340,-115.515,167.145,52.887,159.749
C03293=1018.560,116.590,-115.533,167.148,52.879,159.748
C03294=1018.565,116.838,-115.552,167.151,52.871,159.747
C03295=1018.569,117.088,-115.570,167.153,52.863,159.746
C03296=1018.575,117.337,-115.589,167.156,52.856,159.745
C03297=1018.580,117.587,-115.607,167.160,52.848,159.744
C03298=1018.585,117.835,-115.626,167.163,52.840,159.743
C03299=1018.590,118.086,-115.645,167.165,52.833,159.742
C03300=1018.595,118.334,-115.664,167.168,52.825,159.741
C03301=1018.600,118.584,-115.683,167.171,52.817,159.740
C03302=1018.607,118.940,-115.709,167.176,52.805,159.739
C03303=1018.615,119.298,-115.736,167.179,52.795,159.737
C03304=1018.622,119.654,-115.763,167.183,52.783,159.736
C03305=1018.629,120.011,-115.790,167.188,52.772,159.735
C03306=1018.634,120.261,-115.809,167.191,52.764,159.734
C03307=1018.639,120.510,-115.827,167.194,52.756,159.733
C03308=1018.644,120.759,-115.846,167.197,52.748,159.732
C03309=1018.650,121.008,-115.865,167.200,52.741,159.731
C03310=1018.655,121.258,-115.884,167.203,52.733,159.730
C03311=1018.660,121.506,-115.902,167.206,52.725,159.729
C03312=1018.666,121.756,-115.922,167.209,52.717,159.728
C03313=1018.670,122.005,-115.940,167.212,52.709,159.727
C03314=1018.675,122.217,-115.956,167.214,52.703,159.726
C03315=1018.680,122.429,-115.972,167.217,52.696,159.725
C03316=1018.683,122.641,-115.988,167.220,52.689,159.725
C03317=1018.688,122.852,-116.004,167.222,52.683,159.724
C03318=1018.692,123.065,-116.020,167.224,52.676,159.723
C03319=1018.697,123.277,-116.036,167.227,52.669,159.722
C03320=1018.701,123.488,-116.052,167.230,52.663,159.721
C03321=1018.706,123.700,-116.068,167.232,52.656,159.720
C03322=1018.711,123.949,-116.087,167.236,52.648,159.719
C03323=1018.716,124.198,-116.105,167.238,52.640,159.718
C03324=1018.721,124.448,-116.125,167.241,52.632,159.717
C03325=1018.726,124.697,-116.144,167.245,52.624,159.716
C03326=1018.731,124.947,-116.162,167.247,52.616,159.715
C03327=1018.737,125.196,-116.181,167.250,52.609,159.714
C03328=1018.742,125.444,-116.200,167.254,52.600,159.714
C03329=1018.747,125.694,-116.219,167.256,52.593,159.713
C03330=1018.752,125.943,-116.237,167.259,52.585,159.712
C03331=1018.758,126.193,-116.257,167.263,52.577,159.711
C03332=1018.763,126.441,-116.276,167.265,52.569,159.710
C03333=1018.769,126.691,-116.295,167.268,52.561,159.709
C03334=1018.773,126.940,-116.313,167.272,52.553,159.708
C03335=1018.779,127.190,-116.332,167.275,52.545,159.707
C03336=1018.784,127.438,-116.351,167.278,52.538,159.706
C03337=1018.790,127.688,-116.370,167.281,52.530,159.705
C03338=1018.795,127.936,-116.389,167.284,52.522,159.704
C03339=1018.800,128.187,-116.408,167.287,52.514,159.703
C03340=1018.805,128.436,-116.427,167.290,52.506,159.702
C03341=1018.810,128.685,-116.446,167.293,52.499,159.701
C03342=1018.815,128.934,-116.465,167.296,52.491,159.700
C03343=1018.821,129.183,-116.485,167.300,52.483,159.699
C03344=1018.826,129.433,-116.503,167.302,52.475,159.698
C03345=1018.832,129.682,-116.522,167.306,52.466,159.697
C03346=1018.837,129.931,-116.541,167.309,52.459,159.696
C03347=1018.842,130.180,-116.561,167.311,52.451,159.695
C03348=1018.847,130.429,-116.580,167.314,52.443,159.694
C03349=1018.852,130.679,-116.599,167.318,52.435,159.693
C03350=1018.857,130.928,-116.618,167.321,52.428,159.692
C03351=1018.862,131.177,-116.638,167.323,52.420,159.691
C03352=1018.867,131.426,-116.657,167.327,52.412,159.691
C03353=1018.872,131.676,-116.676,167.330,52.405,159.690
C03354=1018.877,131.925,-116.696,167.333,52.397,159.689
C03355=1018.882,132.174,-116.715,167.337,52.389,159.688
C03356=1018.887,132.423,-116.734,167.339,52.381,159.687
C03357=1018.892,132.672,-116.754,167.342,52.373,159.686
C03358=1018.897,132.922,-116.773,167.345,52.366,159.685
C03359=1018.903,133.170,-116.793,167.349,52.358,159.684
C03360=1018.909,133.420,-116.812,167.352,52.350,159.683
C03361=1018.913,133.669,-116.832,167.354,52.343,159.682
C03362=1018.919,133.918,-116.851,167.358,52.335,159.681
C03363=1018.923,134.167,-116.871,167.361,52.327,159.680
C03364=1018.929,134.417,-116.890,167.364,52.319,159.679
C03365=1018.933,134.666,-116.909,167.368,52.312,159.678
C03366=1018.939,134.915,-116.928,167.371,52.304,159.677
C03367=1018.944,135.165,-116.948,167.373,52.296,159.676
C03368=1018.949,135.413,-116.968,167.377,52.288,159.675
C03369=1018.955,135.662,-116.987,167.380,52.280,159.674
C03370=1018.959,135.912,-117.007,167.383,52.273,159.673
C03371=1018.965,136.161,-117.026,167.386,52.265,159.672
C03372=1018.970,136.411,-117.046,167.389,52.257,159.672
C03373=1018.975,136.659,-117.065,167.392,52.250,159.671
C03374=1018.980,136.909,-117.085,167.396,52.242,159.670
C03375=1018.985,137.157,-117.104,167.399,52.234,159.669
C03376=1018.990,137.407,-117.124,167.401,52.226,159.668
C03377=1018.996,137.656,-117.144,167.405,52.218,159.667
C03378=1019.000,137.905,-117.163,167.408,52.210,159.666
C03379=1019.005,138.155,-117.183,167.412,52.203,159.665
C03380=1019.011,138.404,-117.202,167.415,52.195,159.664
C03381=1019.016,138.652,-117.223,167.418,52.188,159.663
C03382=1019.022,138.935,-117.245,167.421,52.179,159.662
C03383=1019.027,139.217,-117.267,167.424,52.170,159.661
C03384=1019.033,139.499,-117.289,167.429,52.162,159.660
C03385=1019.039,139.781,-117.312,167.433,52.153,159.659
C03386=1019.044,140.031,-117.332,167.435,52.145,159.658
C03387=1019.049,140.279,-117.352,167.438,52.137,159.657
C03388=1019.054,140.529,-117.372,167.442,52.130,159.656
C03389=1019.060,140.778,-117.392,167.445,52.122,159.655
C03390=1019.064,141.027,-117.411,167.448,52.115,159.654
C03391=1019.069,141.276,-117.431,167.452,52.107,159.653
C03392=1019.075,141.525,-117.451,167.454,52.099,159.652
C03393=1019.079,141.774,-117.470,167.459,52.091,159.652
C03394=1019.085,142.023,-117.491,167.461,52.084,159.651
C03395=1019.090,142.273,-117.510,167.464,52.076,159.650
C03396=1019.095,142.521,-117.530,167.468,52.068,159.649
C03397=1019.100,142.771,-117.550,167.471,52.060,159.648
C03398=1019.105,143.020,-117.571,167.474,52.053,159.647
C03399=1019.110,143.269,-117.590,167.478,52.045,159.646
C03400=1019.116,143.518,-117.610,167.481,52.038,159.645
C03401=1019.120,143.768,-117.630,167.484,52.029,159.644
C03402=1019.126,144.017,-117.650,167.487,52.022,159.643
C03403=1019.131,144.266,-117.669,167.490,52.014,159.642
C03404=1019.136,144.515,-117.690,167.494,52.007,159.642
C03405=1019.142,144.764,-117.709,167.497,51.999,159.641
C03406=1019.147,145.013,-117.730,167.501,51.991,159.640
C03407=1019.151,145.262,-117.749,167.504,51.983,159.639
C03408=1019.157,145.511,-117.770,167.506,51.976,159.638
C03409=1019.162,145.761,-117.789,167.510,51.968,159.637
C03410=1019.168,146.010,-117.810,167.513,51.961,159.636
C03411=1019.172,146.258,-117.830,167.517,51.953,159.635
C03412=1019.177,146.508,-117.850,167.520,51.945,159.634
C03413=1019.182,146.757,-117.870,167.523,51.937,159.633
C03414=1019.188,147.006,-117.891,167.527,51.930,159.632
C03415=1019.193,147.256,-117.911,167.530,51.922,159.631
C03416=1019.197,147.505,-117.931,167.533,51.914,159.630
C03417=1019.203,147.754,-117.951,167.536,51.906,159.629
C03418=1019.208,148.003,-117.971,167.540,51.899,159.629
C03419=1019.213,148.252,-117.991,167.544,51.891,159.628
C03420=1019.218,148.501,-118.011,167.546,51.884,159.627
C03421=1019.223,148.750,-118.032,167.550,51.877,159.626
C03422=1019.228,149.000,-118.052,167.553,51.869,159.625
C03423=1019.234,149.249,-118.072,167.556,51.861,159.624
C03424=1019.239,149.498,-118.093,167.560,51.853,159.623
C03425=1019.244,149.747,-118.113,167.563,51.846,159.622
C03426=1019.248,149.996,-118.133,167.566,51.838,159.621
C03427=1019.254,150.245,-118.153,167.570,51.830,159.620
C03428=1019.259,150.494,-118.174,167.573,51.823,159.619
C03429=1019.264,150.743,-118.194,167.577,51.815,159.619
C03430=1019.269,150.992,-118.215,167.580,51.808,159.618
C03431=1019.275,151.242,-118.236,167.583,51.800,159.617
C03432=1019.279,151.491,-118.255,167.586,51.792,159.616
C03433=1019.284,151.740,-118.276,167.590,51.785,159.615
C03434=1019.290,151.989,-118.296,167.594,51.777,159.614
C03435=1019.295,152.238,-118.317,167.596,51.770,159.613
C03436=1019.300,152.487,-118.337,167.600,51.762,159.612
C03437=1019.305,152.736,-118.358,167.604,51.755,159.611
C03438=1019.311,152.985,-118.378,167.607,51.747,159.611
C03439=1019.316,153.235,-118.399,167.610,51.739,159.610
C03440=1019.321,153.483,-118.419,167.613,51.732,159.609
C03441=1019.326,153.732,-118.440,167.617,51.724,159.608
C03442=1019.330,153.982,-118.460,167.620,51.716,159.607
C03443=1019.335,154.231,-118.481,167.624,51.709,159.606
C03444=1019.340,154.480,-118.501,167.627,51.701,159.605
C03445=1019.346,154.729,-118.522,167.630,51.694,159.604
C03446=1019.352,155.011,-118.546,167.635,51.685,159.603
C03447=1019.358,155.292,-118.569,167.638,51.677,159.602
C03448=1019.363,155.575,-118.592,167.642,51.668,159.601
C03449=1019.369,155.857,-118.616,167.646,51.659,159.600
C03450=1019.374,156.106,-118.637,167.650,51.652,159.599
C03451=1019.379,156.355,-118.657,167.654,51.644,159.599
C03452=1019.385,156.604,-118.678,167.656,51.636,159.597
C03453=1019.390,156.854,-118.698,167.661,51.629,159.597
C03454=1019.395,157.103,-118.719,167.664,51.622,159.596
C03455=1019.400,157.351,-118.739,167.666,51.614,159.595
C03456=1019.404,157.601,-118.760,167.671,51.607,159.594
C03457=1019.410,157.850,-118.781,167.674,51.599,159.593
C03458=1019.415,158.099,-118.801,167.677,51.591,159.592
C03459=1019.420,158.347,-118.823,167.680,51.583,159.591
C03460=1019.426,158.596,-118.843,167.685,51.576,159.591
C03461=1019.431,158.846,-118.864,167.687,51.568,159.590
C03462=1019.435,159.095,-118.885,167.692,51.561,159.589
C03463=1019.440,159.344,-118.907,167.695,51.554,159.588
C03464=1019.446,159.593,-118.927,167.698,51.547,159.587
C03465=1019.450,159.842,-118.948,167.702,51.539,159.586
C03466=1019.456,160.091,-118.970,167.705,51.532,159.585
C03467=1019.460,160.340,-118.991,167.709,51.524,159.584
C03468=1019.465,160.589,-119.013,167.712,51.517,159.584
C03469=1019.470,160.838,-119.033,167.715,51.509,159.583
C03470=1019.475,161.088,-119.054,167.719,51.502,159.582
C03471=1019.480,161.337,-119.076,167.722,51.494,159.581
C03472=1019.485,161.586,-119.097,167.727,51.487,159.580
C03473=1019.490,161.834,-119.119,167.729,51.480,159.579
C03474=1019.495,162.084,-119.139,167.733,51.473,159.578
C03475=1019.499,162.333,-119.160,167.737,51.465,159.578
C03476=1019.504,162.582,-119.182,167.740,51.458,159.577
C03477=1019.509,162.831,-119.203,167.744,51.450,159.576
C03478=1019.514,163.080,-119.225,167.747,51.443,159.575
C03479=1019.520,163.329,-119.245,167.751,51.435,159.574
C03480=1019.524,163.578,-119.267,167.754,51.428,159.573
C03481=1019.529,163.827,-119.288,167.757,51.420,159.572
C03482=1019.534,164.076,-119.309,167.762,51.413,159.572
C03483=1019.539,164.325,-119.331,167.764,51.406,159.571
C03484=1019.545,164.574,-119.352,167.769,51.398,159.570
C03485=1019.550,164.824,-119.373,167.772,51.391,159.569
C03486=1019.554,165.073,-119.395,167.776,51.384,159.568
C03487=1019.560,165.321,-119.416,167.779,51.376,159.567
C03488=1019.565,165.570,-119.438,167.783,51.369,159.567
C03489=1019.569,165.819,-119.460,167.786,51.361,159.566
C03490=1019.575,166.068,-119.480,167.790,51.354,159.565
C03491=1019.579,166.317,-119.502,167.793,51.346,159.564
C03492=1019.585,166.566,-119.522,167.798,51.339,159.563
C03493=1019.590,166.815,-119.544,167.801,51.331,159.562
C03494=1019.594,167.064,-119.566,167.805,51.324,159.562
C03495=1019.600,167.314,-119.587,167.808,51.317,159.561
C03496=1019.605,167.563,-119.609,167.812,51.309,159.560
C03497=1019.610,167.812,-119.630,167.815,51.302,159.559
C03498=1019.615,168.061,-119.651,167.819,51.295,159.558
C03499=1019.620,168.309,-119.673,167.822,51.287,159.557
C03500=1019.625,168.558,-119.694,167.827,51.280,159.557
C03501=1019.630,168.807,-119.716,167.830,51.272,159.556
C03502=1019.635,169.057,-119.738,167.834,51.265,159.555
C03503=1019.641,169.306,-119.758,167.838,51.257,159.554
C03504=1019.646,169.555,-119.780,167.841,51.250,159.553
C03505=1019.650,169.804,-119.802,167.845,51.242,159.552
C03506=1019.656,170.053,-119.823,167.849,51.235,159.551
C03507=1019.661,170.302,-119.845,167.852,51.228,159.551
C03508=1019.667,170.551,-119.866,167.856,51.221,159.550
C03509=1019.671,170.800,-119.888,167.860,51.213,159.549
C03510=1019.677,171.082,-119.912,167.864,51.205,159.548
C03511=1019.683,171.363,-119.937,167.868,51.196,159.547
C03512=1019.688,171.645,-119.961,167.872,51.187,159.546
C03513=1019.695,171.927,-119.986,167.877,51.179,159.545
C03514=1019.700,172.176,-120.007,167.880,51.172,159.544
C03515=1019.705,172.425,-120.029,167.884,51.164,159.543
C03516=1019.709,172.673,-120.050,167.888,51.156,159.543
C03517=1019.716,172.923,-120.072,167.891,51.150,159.542
C03518=1019.720,173.171,-120.094,167.895,51.142,159.541
C03519=1019.726,173.421,-120.114,167.899,51.135,159.540
C03520=1019.731,173.669,-120.136,167.903,51.127,159.539
C03521=1019.736,173.919,-120.159,167.907,51.120,159.538
C03522=1019.742,174.167,-120.180,167.910,51.112,159.537
C03523=1019.746,174.416,-120.202,167.914,51.105,159.537
C03524=1019.752,174.666,-120.224,167.918,51.097,159.536
C03525=1019.757,174.915,-120.244,167.922,51.090,159.535
C03526=1019.762,175.164,-120.266,167.926,51.082,159.534
C03527=1019.767,175.413,-120.289,167.930,51.075,159.533
C03528=1019.773,175.662,-120.310,167.933,51.068,159.532
C03529=1019.778,175.910,-120.332,167.937,51.060,159.532
C03530=1019.783,176.160,-120.354,167.941,51.053,159.531
C03531=1019.789,176.408,-120.375,167.944,51.045,159.530
C03532=1019.793,176.657,-120.397,167.949,51.038,159.529
C03533=1019.799,176.907,-120.419,167.953,51.030,159.528
C03534=1019.804,177.155,-120.441,167.956,51.023,159.527
C03535=1019.809,177.404,-120.462,167.960,51.015,159.527
C03536=1019.815,177.654,-120.485,167.964,51.008,159.526
C03537=1019.820,177.902,-120.506,167.968,51.000,159.525
C03538=1019.826,178.152,-120.528,167.971,50.993,159.524
C03539=1019.831,178.400,-120.549,167.976,50.986,159.523
C03540=1019.836,178.649,-120.571,167.980,50.978,159.522
C03541=1019.842,178.898,-120.593,167.983,50.971,159.522
C03542=1019.847,179.147,-120.615,167.987,50.963,159.521
C03543=1019.852,179.397,-120.637,167.991,50.956,159.520
C03544=1019.857,179.645,-120.659,167.995,50.948,159.519
C03545=1019.863,179.894,-120.680,167.999,50.941,159.518
C03546=1019.868,180.143,-120.702,168.003,50.933,159.517
C03547=1019.873,180.392,-120.724,168.007,50.926,159.517
C03548=1019.879,180.641,-120.746,168.011,50.918,159.516
C03549=1019.884,180.890,-120.768,168.015,50.910,159.515
C03550=1019.890,181.140,-120.790,168.018,50.904,159.514
C03551=1019.895,181.388,-120.811,168.022,50.896,159.513
C03552=1019.901,181.638,-120.833,168.027,50.889,159.513
C03553=1019.906,181.886,-120.856,168.031,50.881,159.512
C03554=1019.911,182.135,-120.878,168.034,50.874,159.511
C03555=1019.916,182.384,-120.900,168.039,50.867,159.510
C03556=1019.921,182.634,-120.922,168.043,50.859,159.509
C03557=1019.926,182.882,-120.946,168.046,50.852,159.508
C03558=1019.931,183.132,-120.968,168.050,50.845,159.508
C03559=1019.936,183.380,-120.990,168.055,50.838,159.507
C03560=1019.941,183.630,-121.013,168.058,50.830,159.506
C03561=1019.946,183.878,-121.036,168.062,50.823,159.505
C03562=1019.951,184.127,-121.058,168.066,50.816,159.505
C03563=1019.957,184.376,-121.081,168.070,50.809,159.504
C03564=1019.961,184.625,-121.103,168.074,50.802,159.503
C03565=1019.966,184.874,-121.126,168.077,50.795,159.502
C03566=1019.971,185.123,-121.148,168.082,50.788,159.501
C03567=1019.976,185.372,-121.171,168.086,50.780,159.501
C03568=1019.981,185.621,-121.193,168.090,50.774,159.500
C03569=1019.987,185.869,-121.216,168.094,50.766,159.499
C03570=1019.991,186.119,-121.239,168.098,50.759,159.498
C03571=1019.997,186.368,-121.262,168.101,50.752,159.498
C03572=1020.001,186.616,-121.283,168.106,50.745,159.497
